LIN {X 0,Y 291.922,Z 233.29,A -85,B 0,C 180,E1 -16667.964,E2 -16667.964} C_VEL
LIN {X 0,Y 291.251,Z 221.348,A -85,B 0,C 180,E1 -16668.598,E2 -16668.598} C_VEL
LIN {X 0,Y 291.234,Z 220.005,A -85,B 0,C 180,E1 -16668.691,E2 -16668.691} C_VEL
LIN {X 0,Y 292.711,Z 208.587,A -85,B 0,C 180,E1 -16673.336,E2 -16673.336} C_VEL
LIN {X 0,Y 294.65,Z 197.089,A -85,B 0,C 180,E1 -16678.051,E2 -16678.051} C_VEL
LIN {X 0,Y 294.841,Z 194.228,A -85,B 0,C 180,E1 -16679.249,E2 -16679.249} C_VEL
LIN {X 0,Y 293.186,Z 185.832,A -85,B 0,C 180,E1 -16682.966,E2 -16682.966} C_VEL
LIN {X 0,Y 291.437,Z 176.187,A -85,B 0,C 180,E1 -16687.432,E2 -16687.432} C_VEL
LIN {X 0,Y 291.323,Z 176.194,A -85,B 0,C 180,E1 -16691.595,E2 -16691.595} C_VEL
LIN {X 0,Y 291.344,Z 176.191,A -85,B 0,C 180,E1 -16695.608,E2 -16695.608} C_VEL
LIN {X 0,Y 291.392,Z 176.185,A -85,B 0,C 180,E1 -16699.367,E2 -16699.367} C_VEL
LIN {X 0,Y 291.423,Z 176.182,A -85,B 0,C 180,E1 -16702.922,E2 -16702.922} C_VEL
LIN {X 0,Y 291.334,Z 176.196,A -85,B 0,C 180,E1 -16706.3,E2 -16706.3} C_VEL
LIN {X 0,Y 291.375,Z 176.19,A -85,B 0,C 180,E1 -16710.259,E2 -16710.259} C_VEL
LIN {X 0,Y 291.404,Z 176.185,A -85,B 0,C 180,E1 -16714.271,E2 -16714.271} C_VEL
LIN {X 0,Y 291.362,Z 176.19,A -85,B 0,C 180,E1 -16717.298,E2 -16717.298} C_VEL
LIN {X 0,Y 291.445,Z 176.179,A -85,B 0,C 180,E1 -16720.269,E2 -16720.269} C_VEL
LIN {X 0,Y 291.542,Z 176.166,A -85,B 0,C 180,E1 -16724.623,E2 -16724.623} C_VEL
LIN {X 0,Y 291.524,Z 176.17,A -85,B 0,C 180,E1 -16728.88,E2 -16728.88} C_VEL
LIN {X 0,Y 291.693,Z 176.149,A -85,B 0,C 180,E1 -16731.688,E2 -16731.688} C_VEL
LIN {X 0,Y 291.618,Z 176.157,A -85,B 0,C 180,E1 -16734.468,E2 -16734.468} C_VEL
LIN {X 0,Y 291.88,Z 176.126,A -85,B 0,C 180,E1 -16738.62,E2 -16738.62} C_VEL
LIN {X 0,Y 291.874,Z 176.127,A -85,B 0,C 180,E1 -16741.38,E2 -16741.38} C_VEL
LIN {X 0,Y 291.732,Z 176.146,A -85,B 0,C 180,E1 -16746.918,E2 -16746.918} C_VEL
LIN {X 0,Y 291.616,Z 176.157,A -85,B 0,C 180,E1 -16749.712,E2 -16749.712} C_VEL
LIN {X 0,Y 291.509,Z 176.172,A -85,B 0,C 180,E1 -16753.951,E2 -16753.951} C_VEL
LIN {X 0,Y 291.474,Z 176.176,A -85,B 0,C 180,E1 -16756.819,E2 -16756.819} C_VEL
LIN {X 0,Y 291.438,Z 176.181,A -85,B 0,C 180,E1 -16759.876,E2 -16759.876} C_VEL
LIN {X 0,Y 291.355,Z 176.194,A -85,B 0,C 180,E1 -16764.209,E2 -16764.209} C_VEL
LIN {X 0,Y 291.346,Z 176.191,A -85,B 0,C 180,E1 -16767.279,E2 -16767.279} C_VEL
LIN {X 0,Y 291.308,Z 176.197,A -85,B 0,C 180,E1 -16770.44,E2 -16770.44} C_VEL
LIN {X 0,Y 291.332,Z 176.196,A -85,B 0,C 180,E1 -16773.7,E2 -16773.7} C_VEL
LIN {X 0,Y 291.383,Z 176.188,A -85,B 0,C 180,E1 -16777.26,E2 -16777.26} C_VEL
LIN {X 0,Y 291.34,Z 176.191,A -85,B 0,C 180,E1 -16780.641,E2 -16780.641} C_VEL
LIN {X 0,Y 291.313,Z 176.195,A -85,B 0,C 180,E1 -16784.398,E2 -16784.398} C_VEL
LIN {X 0,Y 291.318,Z 176.194,A -85,B 0,C 180,E1 -16788.406,E2 -16788.406} C_VEL
LIN {X 0,Y 291.345,Z 176.194,A -85,B 0,C 180,E1 -16791.16,E2 -16791.16} C_VEL
LIN {X 0,Y 291.354,Z 176.191,A -85,B 0,C 180,E1 -16794.628,E2 -16794.628} C_VEL
LIN {X 0,Y 291.366,Z 176.188,A -85,B 0,C 180,E1 -16797.953,E2 -16797.953} C_VEL
LIN {X 0,Y 291.378,Z 176.19,A -85,B 0,C 180,E1 -16801.161,E2 -16801.161} C_VEL
LIN {X 0,Y 291.412,Z 176.184,A -85,B 0,C 180,E1 -16804.274,E2 -16804.274} C_VEL
LIN {X 0,Y 291.378,Z 176.187,A -85,B 0,C 180,E1 -16807.302,E2 -16807.302} C_VEL
LIN {X 0,Y 291.455,Z 176.179,A -85,B 0,C 180,E1 -16810.273,E2 -16810.273} C_VEL
LIN {X 0,Y 291.553,Z 176.169,A -85,B 0,C 180,E1 -16814.626,E2 -16814.626} C_VEL
LIN {X 0,Y 291.536,Z 176.168,A -85,B 0,C 180,E1 -16818.883,E2 -16818.883} C_VEL
LIN {X 0,Y 291.709,Z 176.147,A -85,B 0,C 180,E1 -16821.691,E2 -16821.691} C_VEL
LIN {X 0,Y 291.632,Z 176.157,A -85,B 0,C 180,E1 -16824.471,E2 -16824.471} C_VEL
LIN {X 0,Y 291.878,Z 176.126,A -85,B 0,C 180,E1 -16828.622,E2 -16828.622} C_VEL
LIN {X 0,Y 291.877,Z 176.126,A -85,B 0,C 180,E1 -16831.382,E2 -16831.382} C_VEL
LIN {X 0,Y 291.749,Z 176.141,A -85,B 0,C 180,E1 -16836.92,E2 -16836.92} C_VEL
LIN {X 0,Y 291.632,Z 176.16,A -85,B 0,C 180,E1 -16839.714,E2 -16839.714} C_VEL
LIN {X 0,Y 291.526,Z 176.17,A -85,B 0,C 180,E1 -16843.952,E2 -16843.952} C_VEL
LIN {X 0,Y 291.491,Z 176.174,A -85,B 0,C 180,E1 -16846.82,E2 -16846.82} C_VEL
LIN {X 0,Y 291.455,Z 176.178,A -85,B 0,C 180,E1 -16849.877,E2 -16849.877} C_VEL
LIN {X 0,Y 291.33,Z 176.193,A -85,B 0,C 180,E1 -16854.214,E2 -16854.214} C_VEL
LIN {X 0,Y 291.354,Z 176.193,A -85,B 0,C 180,E1 -16857.281,E2 -16857.281} C_VEL
LIN {X 0,Y 291.323,Z 176.194,A -85,B 0,C 180,E1 -16860.441,E2 -16860.441} C_VEL
LIN {X 0,Y 291.349,Z 176.191,A -85,B 0,C 180,E1 -16863.7,E2 -16863.7} C_VEL
LIN {X 0,Y 291.373,Z 176.188,A -85,B 0,C 180,E1 -16867.253,E2 -16867.253} C_VEL
LIN {X 0,Y 291.305,Z 176.201,A -85,B 0,C 180,E1 -16870.649,E2 -16870.649} C_VEL
LIN {X 0,Y 291.288,Z 176.202,A -85,B 0,C 180,E1 -16874.405,E2 -16874.405} C_VEL
LIN {X 0,Y 291.353,Z 176.195,A -85,B 0,C 180,E1 -16878.401,E2 -16878.401} C_VEL
LIN {X 0,Y 291.346,Z 176.191,A -85,B 0,C 180,E1 -16881.157,E2 -16881.157} C_VEL
LIN {X 0,Y 291.506,Z 176.256,A -85,B 0,C 180,E1 -16885.059,E2 -16885.059} C_VEL
LIN {X 0,Y 292.388,Z 181.277,A -85,B 0,C 180,E1 -16888.075,E2 -16888.075} C_VEL
LIN {X 0,Y 292.465,Z 184.403,A -85,B 0,C 180,E1 -16889.896,E2 -16889.896} C_VEL
LIN {X 0,Y 291.785,Z 191.023,A -85,B 0,C 180,E1 -16893.632,E2 -16893.632} C_VEL
LIN {X 0,Y 291.087,Z 198.926,A -85,B 0,C 180,E1 -16898.023,E2 -16898.023} C_VEL
LIN {X 0,Y 290.624,Z 205.588,A -85,B 0,C 180,E1 -16901.677,E2 -16901.677} C_VEL
LIN {X 0,Y 290.148,Z 213.535,A -85,B 0,C 180,E1 -16905.982,E2 -16905.982} C_VEL
LIN {X 0,Y 290.064,Z 216.758,A -85,B 0,C 180,E1 -16907.627,E2 -16907.627} C_VEL
LIN {X 0,Y 290.735,Z 227.966,A -85,B 0,C 180,E1 -16908.496,E2 -16908.496} C_VEL
LIN {X 0,Y 291.517,Z 238.59,A -85,B 0,C 180,E1 -16909.583,E2 -16909.583} C_VEL
LIN {X 0,Y 291.006,Z 247.91,A -85,B 0,C 180,E1 -16910.793,E2 -16910.793} C_VEL
LIN {X 0,Y 290.536,Z 257.449,A -85,B 0,C 180,E1 -16912.355,E2 -16912.355} C_VEL
LIN {X 0,Y 290.137,Z 266.131,A -85,B 0,C 180,E1 -16914.18,E2 -16914.18} C_VEL
LIN {X 0,Y 289.948,Z 272.322,A -85,B 0,C 180,E1 -16915.83,E2 -16915.83} C_VEL
LIN {X 0,Y 289.63,Z 278.288,A -85,B 0,C 180,E1 -16917.914,E2 -16917.914} C_VEL
LIN {X 0,Y 289.621,Z 282.573,A -85,B 0,C 180,E1 -16920,E2 -16920} C_VEL
LIN {X 0,Y 289.778,Z 284.578,A -85,B 0,C 180,E1 -16921.39,E2 -16921.39} C_VEL
LIN {X 0,Y 290.075,Z 285.942,A -85,B 0,C 180,E1 -16922.778,E2 -16922.778} C_VEL
LIN {X 0,Y 290.874,Z 286.751,A -85,B 0,C 180,E1 -16924.841,E2 -16924.841} C_VEL
LIN {X 0,Y 290.556,Z 286.874,A -85,B 0,C 180,E1 -16925.623,E2 -16925.623} C_VEL
LIN {X 0,Y 288.243,Z 286.846,A -85,B 0,C 180,E1 -16926.881,E2 -16926.881} C_VEL
LIN {X 0,Y 285.999,Z 286.418,A -85,B 0,C 180,E1 -16928.153,E2 -16928.153} C_VEL
LIN {X 0,Y 285.799,Z 285.781,A -85,B 0,C 180,E1 -16928.941,E2 -16928.941} C_VEL
LIN {X 0,Y 287.146,Z 283.854,A -85,B 0,C 180,E1 -16930.578,E2 -16930.578} C_VEL
LIN {X 0,Y 289.141,Z 280.078,A -85,B 0,C 180,E1 -16932.636,E2 -16932.636} C_VEL
LIN {X 0,Y 291.713,Z 274.767,A -85,B 0,C 180,E1 -16934.653,E2 -16934.653} C_VEL
LIN {X 0,Y 294.634,Z 267.761,A -85,B 0,C 180,E1 -16936.633,E2 -16936.633} C_VEL
LIN {X 0,Y 296.937,Z 260.933,A -85,B 0,C 180,E1 -16938.173,E2 -16938.173} C_VEL
LIN {X 0,Y 297.396,Z 254.438,A -85,B 0,C 180,E1 -16939.679,E2 -16939.679} C_VEL
LIN {X 0,Y 297.034,Z 246.793,A -85,B 0,C 180,E1 -16941.399,E2 -16941.399} C_VEL
LIN {X 0,Y 295.632,Z 237.751,A -85,B 0,C 180,E1 -16943.44,E2 -16943.44} C_VEL
LIN {X 0,Y 293.399,Z 228.753,A -85,B 0,C 180,E1 -16945.542,E2 -16945.542} C_VEL
LIN {X 0,Y 290.202,Z 219.279,A -85,B 0,C 180,E1 -16947.984,E2 -16947.984} C_VEL
LIN {X 0,Y 290.597,Z 218.071,A -85,B 0,C 180,E1 -16948.927,E2 -16948.927} C_VEL
LIN {X 0,Y 292.066,Z 214.685,A -85,B 0,C 180,E1 -16952.623,E2 -16952.623} C_VEL
LIN {X 0,Y 292.453,Z 212.978,A -85,B 0,C 180,E1 -16955.223,E2 -16955.223} C_VEL
LIN {X 0,Y 292.573,Z 211.549,A -85,B 0,C 180,E1 -16958.65,E2 -16958.65} C_VEL
LIN {X 0,Y 292.684,Z 210.994,A -85,B 0,C 180,E1 -16962.248,E2 -16962.248} C_VEL
LIN {X 0,Y 293.006,Z 211.385,A -85,B 0,C 180,E1 -16966.02,E2 -16966.02} C_VEL
LIN {X 0,Y 293.322,Z 212.845,A -85,B 0,C 180,E1 -16969.688,E2 -16969.688} C_VEL
LIN {X 0,Y 293.711,Z 215.311,A -85,B 0,C 180,E1 -16973.256,E2 -16973.256} C_VEL
LIN {X 0,Y 294.042,Z 216.854,A -85,B 0,C 180,E1 -16974.994,E2 -16974.994} C_VEL
LIN {X 0,Y 294.515,Z 220.412,A -85,B 0,C 180,E1 -16978.166,E2 -16978.166} C_VEL
LIN {X 0,Y 296.581,Z 225.556,A -85,B 0,C 180,E1 -16979.265,E2 -16979.265} C_VEL
LIN {X 0,Y 298.966,Z 236.054,A -85,B 0,C 180,E1 -16981.041,E2 -16981.041} C_VEL
LIN {X 0,Y 300.396,Z 246.753,A -85,B 0,C 180,E1 -16982.753,E2 -16982.753} C_VEL
LIN {X 0,Y 300.603,Z 256.384,A -85,B 0,C 180,E1 -16984.261,E2 -16984.261} C_VEL
LIN {X 0,Y 299.872,Z 262.807,A -85,B 0,C 180,E1 -16985.231,E2 -16985.231} C_VEL
LIN {X 0,Y 297.025,Z 272.375,A -85,B 0,C 180,E1 -16986.649,E2 -16986.649} C_VEL
LIN {X 0,Y 294.133,Z 281.208,A -85,B 0,C 180,E1 -16988.26,E2 -16988.26} C_VEL
LIN {X 0,Y 291.061,Z 289.915,A -85,B 0,C 180,E1 -16990.24,E2 -16990.24} C_VEL
LIN {X 0,Y 288.565,Z 296.948,A -85,B 0,C 180,E1 -16992.274,E2 -16992.274} C_VEL
LIN {X 0,Y 286.676,Z 302.672,A -85,B 0,C 180,E1 -16994.353,E2 -16994.353} C_VEL
LIN {X 0,Y 284.897,Z 307.26,A -85,B 0,C 180,E1 -16996.445,E2 -16996.445} C_VEL
LIN {X 0,Y 283.731,Z 310.784,A -85,B 0,C 180,E1 -16998.569,E2 -16998.569} C_VEL
LIN {X 0,Y 282.79,Z 313.971,A -85,B 0,C 180,E1 -17001.422,E2 -17001.422} C_VEL
LIN {X 0,Y 282.552,Z 314.982,A -85,B 0,C 180,E1 -17002.854,E2 -17002.854} C_VEL
LIN {X 0,Y 282.488,Z 315.573,A -85,B 0,C 180,E1 -17004.362,E2 -17004.362} C_VEL
LIN {X 0,Y 282.48,Z 315.734,A -85,B 0,C 180,E1 -17005.717,E2 -17005.717} C_VEL
LIN {X 0,Y 282.487,Z 315.516,A -85,B 0,C 180,E1 -17007.146,E2 -17007.146} C_VEL
LIN {X 0,Y 282.811,Z 314.871,A -85,B 0,C 180,E1 -17008.574,E2 -17008.574} C_VEL
LIN {X 0,Y 282.89,Z 313.769,A -85,B 0,C 180,E1 -17009.998,E2 -17009.998} C_VEL
LIN {X 0,Y 282.885,Z 311.242,A -85,B 0,C 180,E1 -17012.133,E2 -17012.133} C_VEL
LIN {X 0,Y 282.838,Z 307.581,A -85,B 0,C 180,E1 -17014.273,E2 -17014.273} C_VEL
LIN {X 0,Y 282.952,Z 302.371,A -85,B 0,C 180,E1 -17016.52,E2 -17016.52} C_VEL
LIN {X 0,Y 283.084,Z 296.24,A -85,B 0,C 180,E1 -17018.564,E2 -17018.564} C_VEL
LIN {X 0,Y 283.332,Z 289.589,A -85,B 0,C 180,E1 -17020.358,E2 -17020.358} C_VEL
LIN {X 0,Y 283.815,Z 281.5,A -85,B 0,C 180,E1 -17022.148,E2 -17022.148} C_VEL
LIN {X 0,Y 284.51,Z 271.428,A -85,B 0,C 180,E1 -17023.934,E2 -17023.934} C_VEL
LIN {X 0,Y 285.137,Z 261.442,A -85,B 0,C 180,E1 -17025.362,E2 -17025.362} C_VEL
LIN {X 0,Y 285.939,Z 250.048,A -85,B 0,C 180,E1 -17026.642,E2 -17026.642} C_VEL
LIN {X 0,Y 285.956,Z 246.019,A -85,B 0,C 180,E1 -17027.023,E2 -17027.023} C_VEL
LIN {X 0,Y 284.874,Z 234.213,A -85,B 0,C 180,E1 -17027.959,E2 -17027.959} C_VEL
LIN {X 0,Y 284.188,Z 222.921,A -85,B 0,C 180,E1 -17028.61,E2 -17028.61} C_VEL
LIN {X 0,Y 284.168,Z 220.049,A -85,B 0,C 180,E1 -17028.752,E2 -17028.752} C_VEL
LIN {X 0,Y 285.522,Z 209.459,A -85,B 0,C 180,E1 -17033.19,E2 -17033.19} C_VEL
LIN {X 0,Y 287.384,Z 198.799,A -85,B 0,C 180,E1 -17037.684,E2 -17037.684} C_VEL
LIN {X 0,Y 287.805,Z 195.191,A -85,B 0,C 180,E1 -17039.232,E2 -17039.232} C_VEL
LIN {X 0,Y 286.013,Z 186.137,A -85,B 0,C 180,E1 -17043.336,E2 -17043.336} C_VEL
LIN {X 0,Y 284.369,Z 177.068,A -85,B 0,C 180,E1 -17047.687,E2 -17047.687} C_VEL
LIN {X 0,Y 284.275,Z 177.073,A -85,B 0,C 180,E1 -17052.125,E2 -17052.125} C_VEL
LIN {X 0,Y 284.31,Z 177.07,A -85,B 0,C 180,E1 -17056.199,E2 -17056.199} C_VEL
LIN {X 0,Y 284.342,Z 177.066,A -85,B 0,C 180,E1 -17060.011,E2 -17060.011} C_VEL
LIN {X 0,Y 284.345,Z 177.064,A -85,B 0,C 180,E1 -17063.616,E2 -17063.616} C_VEL
LIN {X 0,Y 284.297,Z 177.069,A -85,B 0,C 180,E1 -17067.188,E2 -17067.188} C_VEL
LIN {X 0,Y 284.347,Z 177.065,A -85,B 0,C 180,E1 -17070.375,E2 -17070.375} C_VEL
LIN {X 0,Y 284.366,Z 177.062,A -85,B 0,C 180,E1 -17073.585,E2 -17073.585} C_VEL
LIN {X 0,Y 284.321,Z 177.066,A -85,B 0,C 180,E1 -17076.703,E2 -17076.703} C_VEL
LIN {X 0,Y 284.39,Z 177.059,A -85,B 0,C 180,E1 -17081.261,E2 -17081.261} C_VEL
LIN {X 0,Y 284.479,Z 177.046,A -85,B 0,C 180,E1 -17084.458,E2 -17084.458} C_VEL
LIN {X 0,Y 284.476,Z 177.047,A -85,B 0,C 180,E1 -17088.601,E2 -17088.601} C_VEL
LIN {X 0,Y 284.643,Z 177.028,A -85,B 0,C 180,E1 -17091.481,E2 -17091.481} C_VEL
LIN {X 0,Y 284.588,Z 177.033,A -85,B 0,C 180,E1 -17094.331,E2 -17094.331} C_VEL
LIN {X 0,Y 284.846,Z 177.002,A -85,B 0,C 180,E1 -17098.586,E2 -17098.586} C_VEL
LIN {X 0,Y 284.84,Z 177.003,A -85,B 0,C 180,E1 -17101.414,E2 -17101.414} C_VEL
LIN {X 0,Y 284.684,Z 177.022,A -85,B 0,C 180,E1 -17107.09,E2 -17107.09} C_VEL
LIN {X 0,Y 284.553,Z 177.037,A -85,B 0,C 180,E1 -17109.956,E2 -17109.956} C_VEL
LIN {X 0,Y 284.469,Z 177.051,A -85,B 0,C 180,E1 -17114.303,E2 -17114.303} C_VEL
LIN {X 0,Y 284.413,Z 177.054,A -85,B 0,C 180,E1 -17117.249,E2 -17117.249} C_VEL
LIN {X 0,Y 284.366,Z 177.064,A -85,B 0,C 180,E1 -17120.243,E2 -17120.243} C_VEL
LIN {X 0,Y 284.314,Z 177.069,A -85,B 0,C 180,E1 -17123.857,E2 -17123.857} C_VEL
LIN {X 0,Y 284.276,Z 177.076,A -85,B 0,C 180,E1 -17128.017,E2 -17128.017} C_VEL
LIN {X 0,Y 284.273,Z 177.073,A -85,B 0,C 180,E1 -17131.277,E2 -17131.277} C_VEL
LIN {X 0,Y 284.351,Z 177.063,A -85,B 0,C 180,E1 -17135.356,E2 -17135.356} C_VEL
LIN {X 0,Y 284.313,Z 177.069,A -85,B 0,C 180,E1 -17138.169,E2 -17138.169} C_VEL
LIN {X 0,Y 284.286,Z 177.07,A -85,B 0,C 180,E1 -17142.132,E2 -17142.132} C_VEL
LIN {X 0,Y 284.26,Z 177.074,A -85,B 0,C 180,E1 -17146.194,E2 -17146.194} C_VEL
LIN {X 0,Y 284.298,Z 177.069,A -85,B 0,C 180,E1 -17150.026,E2 -17150.026} C_VEL
LIN {X 0,Y 284.325,Z 177.067,A -85,B 0,C 180,E1 -17153.616,E2 -17153.616} C_VEL
LIN {X 0,Y 284.301,Z 177.072,A -85,B 0,C 180,E1 -17157.192,E2 -17157.192} C_VEL
LIN {X 0,Y 284.353,Z 177.061,A -85,B 0,C 180,E1 -17160.378,E2 -17160.378} C_VEL
LIN {X 0,Y 284.373,Z 177.06,A -85,B 0,C 180,E1 -17163.589,E2 -17163.589} C_VEL
LIN {X 0,Y 284.363,Z 177.065,A -85,B 0,C 180,E1 -17166.709,E2 -17166.709} C_VEL
LIN {X 0,Y 284.401,Z 177.057,A -85,B 0,C 180,E1 -17171.264,E2 -17171.264} C_VEL
LIN {X 0,Y 284.49,Z 177.05,A -85,B 0,C 180,E1 -17174.461,E2 -17174.461} C_VEL
LIN {X 0,Y 284.487,Z 177.048,A -85,B 0,C 180,E1 -17178.604,E2 -17178.604} C_VEL
LIN {X 0,Y 284.659,Z 177.024,A -85,B 0,C 180,E1 -17181.483,E2 -17181.483} C_VEL
LIN {X 0,Y 284.602,Z 177.034,A -85,B 0,C 180,E1 -17184.334,E2 -17184.334} C_VEL
LIN {X 0,Y 284.846,Z 177.002,A -85,B 0,C 180,E1 -17188.588,E2 -17188.588} C_VEL
LIN {X 0,Y 284.845,Z 177.002,A -85,B 0,C 180,E1 -17191.416,E2 -17191.416} C_VEL
LIN {X 0,Y 284.701,Z 177.019,A -85,B 0,C 180,E1 -17197.092,E2 -17197.092} C_VEL
LIN {X 0,Y 284.57,Z 177.037,A -85,B 0,C 180,E1 -17199.957,E2 -17199.957} C_VEL
LIN {X 0,Y 284.485,Z 177.045,A -85,B 0,C 180,E1 -17204.305,E2 -17204.305} C_VEL
LIN {X 0,Y 284.429,Z 177.056,A -85,B 0,C 180,E1 -17207.25,E2 -17207.25} C_VEL
LIN {X 0,Y 284.38,Z 177.058,A -85,B 0,C 180,E1 -17210.244,E2 -17210.244} C_VEL
LIN {X 0,Y 284.287,Z 177.073,A -85,B 0,C 180,E1 -17214.853,E2 -17214.853} C_VEL
LIN {X 0,Y 284.285,Z 177.07,A -85,B 0,C 180,E1 -17218.018,E2 -17218.018} C_VEL
LIN {X 0,Y 284.29,Z 177.072,A -85,B 0,C 180,E1 -17221.277,E2 -17221.277} C_VEL
LIN {X 0,Y 284.342,Z 177.065,A -85,B 0,C 180,E1 -17225.348,E2 -17225.348} C_VEL
LIN {X 0,Y 284.306,Z 177.068,A -85,B 0,C 180,E1 -17228.172,E2 -17228.172} C_VEL
LIN {X 0,Y 284.242,Z 177.077,A -85,B 0,C 180,E1 -17232.118,E2 -17232.118} C_VEL
LIN {X 0,Y 284.262,Z 177.076,A -85,B 0,C 180,E1 -17236.19,E2 -17236.19} C_VEL
LIN {X 0,Y 284.313,Z 177.069,A -85,B 0,C 180,E1 -17240.025,E2 -17240.025} C_VEL
LIN {X 0,Y 284.437,Z 177.055,A -85,B 0,C 180,E1 -17244.628,E2 -17244.628} C_VEL
LIN {X 0,Y 284.477,Z 177.176,A -85,B 0,C 180,E1 -17245.005,E2 -17245.005} C_VEL
LIN {X 0,Y 285.355,Z 182.094,A -85,B 0,C 180,E1 -17248.027,E2 -17248.027} C_VEL
LIN {X 0,Y 285.462,Z 184.594,A -85,B 0,C 180,E1 -17249.51,E2 -17249.51} C_VEL
LIN {X 0,Y 284.918,Z 190.002,A -85,B 0,C 180,E1 -17252.627,E2 -17252.627} C_VEL
LIN {X 0,Y 284.191,Z 197.115,A -85,B 0,C 180,E1 -17256.692,E2 -17256.692} C_VEL
LIN {X 0,Y 283.715,Z 203.489,A -85,B 0,C 180,E1 -17260.277,E2 -17260.277} C_VEL
LIN {X 0,Y 283.189,Z 210.47,A -85,B 0,C 180,E1 -17264.158,E2 -17264.158} C_VEL
LIN {X 0,Y 283,Z 216.617,A -85,B 0,C 180,E1 -17267.541,E2 -17267.541} C_VEL
LIN {X 0,Y 283.653,Z 228.157,A -85,B 0,C 180,E1 -17268.477,E2 -17268.477} C_VEL
LIN {X 0,Y 284.437,Z 237.98,A -85,B 0,C 180,E1 -17269.501,E2 -17269.501} C_VEL
LIN {X 0,Y 283.903,Z 248.683,A -85,B 0,C 180,E1 -17270.92,E2 -17270.92} C_VEL
LIN {X 0,Y 283.387,Z 258.077,A -85,B 0,C 180,E1 -17272.519,E2 -17272.519} C_VEL
LIN {X 0,Y 283.042,Z 266.311,A -85,B 0,C 180,E1 -17274.3,E2 -17274.3} C_VEL
LIN {X 0,Y 282.815,Z 272.827,A -85,B 0,C 180,E1 -17276.082,E2 -17276.082} C_VEL
LIN {X 0,Y 282.552,Z 277.884,A -85,B 0,C 180,E1 -17277.862,E2 -17277.862} C_VEL
LIN {X 0,Y 282.533,Z 282.42,A -85,B 0,C 180,E1 -17280,E2 -17280} C_VEL
LIN {X 0,Y 282.69,Z 284.584,A -85,B 0,C 180,E1 -17281.425,E2 -17281.425} C_VEL
LIN {X 0,Y 282.992,Z 286.121,A -85,B 0,C 180,E1 -17282.847,E2 -17282.847} C_VEL
LIN {X 0,Y 283.491,Z 287.052,A -85,B 0,C 180,E1 -17284.265,E2 -17284.265} C_VEL
LIN {X 0,Y 284.199,Z 287.358,A -85,B 0,C 180,E1 -17285.677,E2 -17285.677} C_VEL
LIN {X 0,Y 284.689,Z 287.086,A -85,B 0,C 180,E1 -17287.09,E2 -17287.09} C_VEL
LIN {X 0,Y 285.799,Z 285.781,A -85,B 0,C 180,E1 -17288.941,E2 -17288.941} C_VEL
LIN {X 0,Y 285.691,Z 285.122,A -85,B 0,C 180,E1 -17289.734,E2 -17289.734} C_VEL
LIN {X 0,Y 282.327,Z 282.599,A -85,B 0,C 180,E1 -17292.33,E2 -17292.33} C_VEL
LIN {X 0,Y 282.538,Z 281.272,A -85,B 0,C 180,E1 -17293.086,E2 -17293.086} C_VEL
LIN {X 0,Y 285.045,Z 276.665,A -85,B 0,C 180,E1 -17295.004,E2 -17295.004} C_VEL
LIN {X 0,Y 288.099,Z 270.13,A -85,B 0,C 180,E1 -17297.022,E2 -17297.022} C_VEL
LIN {X 0,Y 290.746,Z 263.4,A -85,B 0,C 180,E1 -17298.654,E2 -17298.654} C_VEL
LIN {X 0,Y 291.479,Z 256.132,A -85,B 0,C 180,E1 -17300.463,E2 -17300.463} C_VEL
LIN {X 0,Y 291.291,Z 248.612,A -85,B 0,C 180,E1 -17302.287,E2 -17302.287} C_VEL
LIN {X 0,Y 290.188,Z 240.323,A -85,B 0,C 180,E1 -17304.313,E2 -17304.313} C_VEL
LIN {X 0,Y 288.364,Z 232.193,A -85,B 0,C 180,E1 -17306.41,E2 -17306.41} C_VEL
LIN {X 0,Y 286.087,Z 224.218,A -85,B 0,C 180,E1 -17308.622,E2 -17308.622} C_VEL
LIN {X 0,Y 284.723,Z 220.89,A -85,B 0,C 180,E1 -17309.733,E2 -17309.733} C_VEL
LIN {X 0,Y 284.378,Z 219.142,A -85,B 0,C 180,E1 -17310.236,E2 -17310.236} C_VEL
LIN {X 0,Y 285.458,Z 216.716,A -85,B 0,C 180,E1 -17313.164,E2 -17313.164} C_VEL
LIN {X 0,Y 285.828,Z 215.025,A -85,B 0,C 180,E1 -17316.166,E2 -17316.166} C_VEL
LIN {X 0,Y 285.928,Z 214.262,A -85,B 0,C 180,E1 -17318.133,E2 -17318.133} C_VEL
LIN {X 0,Y 286.043,Z 213.65,A -85,B 0,C 180,E1 -17321.559,E2 -17321.559} C_VEL
LIN {X 0,Y 286.337,Z 213.883,A -85,B 0,C 180,E1 -17325.381,E2 -17325.381} C_VEL
LIN {X 0,Y 286.589,Z 214.93,A -85,B 0,C 180,E1 -17328.536,E2 -17328.536} C_VEL
LIN {X 0,Y 286.995,Z 217.115,A -85,B 0,C 180,E1 -17332.249,E2 -17332.249} C_VEL
LIN {X 0,Y 287.243,Z 218.52,A -85,B 0,C 180,E1 -17334.038,E2 -17334.038} C_VEL
LIN {X 0,Y 287.531,Z 220.433,A -85,B 0,C 180,E1 -17335.912,E2 -17335.912} C_VEL
LIN {X 0,Y 289.002,Z 223.556,A -85,B 0,C 180,E1 -17336.801,E2 -17336.801} C_VEL
LIN {X 0,Y 290.855,Z 226.417,A -85,B 0,C 180,E1 -17337.749,E2 -17337.749} C_VEL
LIN {X 0,Y 292.337,Z 230.74,A -85,B 0,C 180,E1 -17338.724,E2 -17338.724} C_VEL
LIN {X 0,Y 294.003,Z 239.669,A -85,B 0,C 180,E1 -17340.356,E2 -17340.356} C_VEL
LIN {X 0,Y 294.981,Z 250.459,A -85,B 0,C 180,E1 -17342.21,E2 -17342.21} C_VEL
LIN {X 0,Y 294.835,Z 259.143,A -85,B 0,C 180,E1 -17343.672,E2 -17343.672} C_VEL
LIN {X 0,Y 294.024,Z 264.385,A -85,B 0,C 180,E1 -17344.514,E2 -17344.514} C_VEL
LIN {X 0,Y 290.713,Z 274.484,A -85,B 0,C 180,E1 -17346.111,E2 -17346.111} C_VEL
LIN {X 0,Y 287.117,Z 284.315,A -85,B 0,C 180,E1 -17348.079,E2 -17348.079} C_VEL
LIN {X 0,Y 283.879,Z 292.575,A -85,B 0,C 180,E1 -17350.181,E2 -17350.181} C_VEL
LIN {X 0,Y 281.17,Z 299.723,A -85,B 0,C 180,E1 -17352.543,E2 -17352.543} C_VEL
LIN {X 0,Y 279.192,Z 304.781,A -85,B 0,C 180,E1 -17354.672,E2 -17354.672} C_VEL
LIN {X 0,Y 277.478,Z 308.764,A -85,B 0,C 180,E1 -17356.821,E2 -17356.821} C_VEL
LIN {X 0,Y 276.162,Z 312.519,A -85,B 0,C 180,E1 -17359.736,E2 -17359.736} C_VEL
LIN {X 0,Y 275.732,Z 313.804,A -85,B 0,C 180,E1 -17361.201,E2 -17361.201} C_VEL
LIN {X 0,Y 275.392,Z 315.135,A -85,B 0,C 180,E1 -17364.139,E2 -17364.139} C_VEL
LIN {X 0,Y 275.401,Z 315.223,A -85,B 0,C 180,E1 -17365.607,E2 -17365.607} C_VEL
LIN {X 0,Y 275.414,Z 314.858,A -85,B 0,C 180,E1 -17367.072,E2 -17367.072} C_VEL
LIN {X 0,Y 275.749,Z 314.114,A -85,B 0,C 180,E1 -17368.537,E2 -17368.537} C_VEL
LIN {X 0,Y 275.84,Z 312.928,A -85,B 0,C 180,E1 -17369.998,E2 -17369.998} C_VEL
LIN {X 0,Y 275.855,Z 310.221,A -85,B 0,C 180,E1 -17372.188,E2 -17372.188} C_VEL
LIN {X 0,Y 275.839,Z 306.336,A -85,B 0,C 180,E1 -17374.381,E2 -17374.381} C_VEL
LIN {X 0,Y 275.932,Z 301.068,A -85,B 0,C 180,E1 -17376.619,E2 -17376.619} C_VEL
LIN {X 0,Y 276.069,Z 294.528,A -85,B 0,C 180,E1 -17378.784,E2 -17378.784} C_VEL
LIN {X 0,Y 276.442,Z 286.025,A -85,B 0,C 180,E1 -17380.99,E2 -17380.99} C_VEL
LIN {X 0,Y 276.948,Z 277.211,A -85,B 0,C 180,E1 -17382.827,E2 -17382.827} C_VEL
LIN {X 0,Y 277.559,Z 268.569,A -85,B 0,C 180,E1 -17384.29,E2 -17384.29} C_VEL
LIN {X 0,Y 278.298,Z 257.965,A -85,B 0,C 180,E1 -17385.749,E2 -17385.749} C_VEL
LIN {X 0,Y 278.952,Z 248.24,A -85,B 0,C 180,E1 -17386.821,E2 -17386.821} C_VEL
LIN {X 0,Y 277.94,Z 236.194,A -85,B 0,C 180,E1 -17387.851,E2 -17387.851} C_VEL
LIN {X 0,Y 277.142,Z 223.946,A -85,B 0,C 180,E1 -17388.622,E2 -17388.622} C_VEL
LIN {X 0,Y 277.097,Z 219.923,A -85,B 0,C 180,E1 -17388.865,E2 -17388.865} C_VEL
LIN {X 0,Y 278.656,Z 208.529,A -85,B 0,C 180,E1 -17393.797,E2 -17393.797} C_VEL
LIN {X 0,Y 280.582,Z 197.88,A -85,B 0,C 180,E1 -17398.416,E2 -17398.416} C_VEL
LIN {X 0,Y 280.71,Z 195.779,A -85,B 0,C 180,E1 -17399.346,E2 -17399.346} C_VEL
LIN {X 0,Y 279.255,Z 188.492,A -85,B 0,C 180,E1 -17402.755,E2 -17402.755} C_VEL
LIN {X 0,Y 277.498,Z 178.813,A -85,B 0,C 180,E1 -17407.429,E2 -17407.429} C_VEL
LIN {X 0,Y 277.304,Z 177.949,A -85,B 0,C 180,E1 -17407.964,E2 -17407.964} C_VEL
LIN {X 0,Y 277.225,Z 177.954,A -85,B 0,C 180,E1 -17412.677,E2 -17412.677} C_VEL
LIN {X 0,Y 277.254,Z 177.947,A -85,B 0,C 180,E1 -17416.81,E2 -17416.81} C_VEL
LIN {X 0,Y 277.258,Z 177.948,A -85,B 0,C 180,E1 -17420.676,E2 -17420.676} C_VEL
LIN {X 0,Y 277.295,Z 177.944,A -85,B 0,C 180,E1 -17424.343,E2 -17424.343} C_VEL
LIN {X 0,Y 277.234,Z 177.951,A -85,B 0,C 180,E1 -17427.835,E2 -17427.835} C_VEL
LIN {X 0,Y 277.26,Z 177.946,A -85,B 0,C 180,E1 -17431.209,E2 -17431.209} C_VEL
LIN {X 0,Y 277.298,Z 177.941,A -85,B 0,C 180,E1 -17434.478,E2 -17434.478} C_VEL
LIN {X 0,Y 277.256,Z 177.95,A -85,B 0,C 180,E1 -17437.652,E2 -17437.652} C_VEL
LIN {X 0,Y 277.332,Z 177.937,A -85,B 0,C 180,E1 -17440.765,E2 -17440.765} C_VEL
LIN {X 0,Y 277.422,Z 177.928,A -85,B 0,C 180,E1 -17445.325,E2 -17445.325} C_VEL
LIN {X 0,Y 277.494,Z 177.917,A -85,B 0,C 180,E1 -17449.788,E2 -17449.788} C_VEL
LIN {X 0,Y 277.636,Z 177.899,A -85,B 0,C 180,E1 -17452.729,E2 -17452.729} C_VEL
LIN {X 0,Y 277.812,Z 177.878,A -85,B 0,C 180,E1 -17458.55,E2 -17458.55} C_VEL
LIN {X 0,Y 277.806,Z 177.879,A -85,B 0,C 180,E1 -17461.45,E2 -17461.45} C_VEL
LIN {X 0,Y 277.639,Z 177.899,A -85,B 0,C 180,E1 -17467.271,E2 -17467.271} C_VEL
LIN {X 0,Y 277.494,Z 177.917,A -85,B 0,C 180,E1 -17470.212,E2 -17470.212} C_VEL
LIN {X 0,Y 277.422,Z 177.929,A -85,B 0,C 180,E1 -17474.675,E2 -17474.675} C_VEL
LIN {X 0,Y 277.334,Z 177.936,A -85,B 0,C 180,E1 -17479.235,E2 -17479.235} C_VEL
LIN {X 0,Y 277.275,Z 177.946,A -85,B 0,C 180,E1 -17483.925,E2 -17483.925} C_VEL
LIN {X 0,Y 277.261,Z 177.946,A -85,B 0,C 180,E1 -17487.486,E2 -17487.486} C_VEL
LIN {X 0,Y 277.236,Z 177.95,A -85,B 0,C 180,E1 -17490.474,E2 -17490.474} C_VEL
LIN {X 0,Y 277.242,Z 177.951,A -85,B 0,C 180,E1 -17493.896,E2 -17493.896} C_VEL
LIN {X 0,Y 277.27,Z 177.947,A -85,B 0,C 180,E1 -17497.469,E2 -17497.469} C_VEL
LIN {X 0,Y 277.217,Z 177.953,A -85,B 0,C 180,E1 -17501.235,E2 -17501.235} C_VEL
LIN {X 0,Y 277.211,Z 177.954,A -85,B 0,C 180,E1 -17505.224,E2 -17505.224} C_VEL
LIN {X 0,Y 277.215,Z 177.954,A -85,B 0,C 180,E1 -17509.514,E2 -17509.514} C_VEL
LIN {X 0,Y 277.26,Z 177.945,A -85,B 0,C 180,E1 -17512.533,E2 -17512.533} C_VEL
LIN {X 0,Y 277.24,Z 177.948,A -85,B 0,C 180,E1 -17516.107,E2 -17516.107} C_VEL
LIN {X 0,Y 277.256,Z 177.946,A -85,B 0,C 180,E1 -17519.541,E2 -17519.541} C_VEL
LIN {X 0,Y 277.354,Z 177.938,A -85,B 0,C 180,E1 -17522.867,E2 -17522.867} C_VEL
LIN {X 0,Y 277.325,Z 177.938,A -85,B 0,C 180,E1 -17526.082,E2 -17526.082} C_VEL
LIN {X 0,Y 277.342,Z 177.939,A -85,B 0,C 180,E1 -17530.769,E2 -17530.769} C_VEL
LIN {X 0,Y 277.433,Z 177.924,A -85,B 0,C 180,E1 -17535.328,E2 -17535.328} C_VEL
LIN {X 0,Y 277.506,Z 177.916,A -85,B 0,C 180,E1 -17539.791,E2 -17539.791} C_VEL
LIN {X 0,Y 277.654,Z 177.898,A -85,B 0,C 180,E1 -17542.732,E2 -17542.732} C_VEL
LIN {X 0,Y 277.813,Z 177.878,A -85,B 0,C 180,E1 -17548.553,E2 -17548.553} C_VEL
LIN {X 0,Y 277.812,Z 177.878,A -85,B 0,C 180,E1 -17551.452,E2 -17551.452} C_VEL
LIN {X 0,Y 277.656,Z 177.898,A -85,B 0,C 180,E1 -17557.273,E2 -17557.273} C_VEL
LIN {X 0,Y 277.51,Z 177.915,A -85,B 0,C 180,E1 -17560.213,E2 -17560.213} C_VEL
LIN {X 0,Y 277.438,Z 177.923,A -85,B 0,C 180,E1 -17564.676,E2 -17564.676} C_VEL
LIN {X 0,Y 277.349,Z 177.938,A -85,B 0,C 180,E1 -17569.236,E2 -17569.236} C_VEL
LIN {X 0,Y 277.259,Z 177.946,A -85,B 0,C 180,E1 -17573.929,E2 -17573.929} C_VEL
LIN {X 0,Y 277.271,Z 177.946,A -85,B 0,C 180,E1 -17577.483,E2 -17577.483} C_VEL
LIN {X 0,Y 277.253,Z 177.946,A -85,B 0,C 180,E1 -17580.474,E2 -17580.474} C_VEL
LIN {X 0,Y 277.251,Z 177.947,A -85,B 0,C 180,E1 -17583.897,E2 -17583.897} C_VEL
LIN {X 0,Y 277.265,Z 177.944,A -85,B 0,C 180,E1 -17587.472,E2 -17587.472} C_VEL
LIN {X 0,Y 277.189,Z 177.955,A -85,B 0,C 180,E1 -17591.243,E2 -17591.243} C_VEL
LIN {X 0,Y 277.204,Z 177.953,A -85,B 0,C 180,E1 -17595.228,E2 -17595.228} C_VEL
LIN {X 0,Y 277.226,Z 177.952,A -85,B 0,C 180,E1 -17598.766,E2 -17598.766} C_VEL
LIN {X 0,Y 277.283,Z 177.945,A -85,B 0,C 180,E1 -17602.533,E2 -17602.533} C_VEL
LIN {X 0,Y 277.405,Z 178.04,A -85,B 0,C 180,E1 -17604.916,E2 -17604.916} C_VEL
LIN {X 0,Y 278.298,Z 182.904,A -85,B 0,C 180,E1 -17607.973,E2 -17607.973} C_VEL
LIN {X 0,Y 278.365,Z 185.703,A -85,B 0,C 180,E1 -17609.672,E2 -17609.672} C_VEL
LIN {X 0,Y 277.794,Z 191.194,A -85,B 0,C 180,E1 -17612.91,E2 -17612.91} C_VEL
LIN {X 0,Y 276.98,Z 199.319,A -85,B 0,C 180,E1 -17617.629,E2 -17617.629} C_VEL
LIN {X 0,Y 276.455,Z 206.021,A -85,B 0,C 180,E1 -17621.472,E2 -17621.472} C_VEL
LIN {X 0,Y 275.967,Z 214.125,A -85,B 0,C 180,E1 -17626.058,E2 -17626.058} C_VEL
LIN {X 0,Y 275.919,Z 216.679,A -85,B 0,C 180,E1 -17627.496,E2 -17627.496} C_VEL
LIN {X 0,Y 276.552,Z 228.21,A -85,B 0,C 180,E1 -17628.456,E2 -17628.456} C_VEL
LIN {X 0,Y 277.286,Z 238.792,A -85,B 0,C 180,E1 -17629.596,E2 -17629.596} C_VEL
LIN {X 0,Y 276.76,Z 249.322,A -85,B 0,C 180,E1 -17631.052,E2 -17631.052} C_VEL
LIN {X 0,Y 276.255,Z 258.627,A -85,B 0,C 180,E1 -17632.692,E2 -17632.692} C_VEL
LIN {X 0,Y 275.954,Z 266.803,A -85,B 0,C 180,E1 -17634.52,E2 -17634.52} C_VEL
LIN {X 0,Y 275.687,Z 273.272,A -85,B 0,C 180,E1 -17636.346,E2 -17636.346} C_VEL
LIN {X 0,Y 275.435,Z 279.193,A -85,B 0,C 180,E1 -17638.538,E2 -17638.538} C_VEL
LIN {X 0,Y 275.502,Z 283.47,A -85,B 0,C 180,E1 -17640.731,E2 -17640.731} C_VEL
LIN {X 0,Y 275.912,Z 286.255,A -85,B 0,C 180,E1 -17642.92,E2 -17642.92} C_VEL
LIN {X 0,Y 276.419,Z 287.339,A -85,B 0,C 180,E1 -17644.375,E2 -17644.375} C_VEL
LIN {X 0,Y 277.146,Z 287.827,A -85,B 0,C 180,E1 -17645.822,E2 -17645.822} C_VEL
LIN {X 0,Y 277.693,Z 287.762,A -85,B 0,C 180,E1 -17647.27,E2 -17647.27} C_VEL
LIN {X 0,Y 278.869,Z 286.686,A -85,B 0,C 180,E1 -17649.17,E2 -17649.17} C_VEL
LIN {X 0,Y 279.574,Z 285.846,A -85,B 0,C 180,E1 -17650.135,E2 -17650.135} C_VEL
LIN {X 0,Y 281.62,Z 282.866,A -85,B 0,C 180,E1 -17652.247,E2 -17652.247} C_VEL
LIN {X 0,Y 282.538,Z 281.272,A -85,B 0,C 180,E1 -17653.086,E2 -17653.086} C_VEL
LIN {X 0,Y 282.819,Z 279.854,A -85,B 0,C 180,E1 -17653.843,E2 -17653.843} C_VEL
LIN {X 0,Y 280.544,Z 275.449,A -85,B 0,C 180,E1 -17656.407,E2 -17656.407} C_VEL
LIN {X 0,Y 280.996,Z 273.519,A -85,B 0,C 180,E1 -17657.109,E2 -17657.109} C_VEL
LIN {X 0,Y 284.437,Z 266.166,A -85,B 0,C 180,E1 -17659.083,E2 -17659.083} C_VEL
LIN {X 0,Y 285.478,Z 260.194,A -85,B 0,C 180,E1 -17660.687,E2 -17660.687} C_VEL
LIN {X 0,Y 285.716,Z 252.319,A -85,B 0,C 180,E1 -17662.746,E2 -17662.746} C_VEL
LIN {X 0,Y 285.066,Z 244.652,A -85,B 0,C 180,E1 -17664.779,E2 -17664.779} C_VEL
LIN {X 0,Y 283.473,Z 235.872,A -85,B 0,C 180,E1 -17667.24,E2 -17667.24} C_VEL
LIN {X 0,Y 281.888,Z 229.238,A -85,B 0,C 180,E1 -17669.233,E2 -17669.233} C_VEL
LIN {X 0,Y 280.752,Z 225.281,A -85,B 0,C 180,E1 -17670.555,E2 -17670.555} C_VEL
LIN {X 0,Y 279.004,Z 220.911,A -85,B 0,C 180,E1 -17672.363,E2 -17672.363} C_VEL
LIN {X 0,Y 278.728,Z 219.345,A -85,B 0,C 180,E1 -17672.903,E2 -17672.903} C_VEL
LIN {X 0,Y 279.219,Z 217.482,A -85,B 0,C 180,E1 -17676.344,E2 -17676.344} C_VEL
LIN {X 0,Y 279.329,Z 216.65,A -85,B 0,C 180,E1 -17678.977,E2 -17678.977} C_VEL
LIN {X 0,Y 279.438,Z 216.31,A -85,B 0,C 180,E1 -17681.014,E2 -17681.014} C_VEL
LIN {X 0,Y 279.684,Z 216.405,A -85,B 0,C 180,E1 -17684.716,E2 -17684.716} C_VEL
LIN {X 0,Y 279.903,Z 217.069,A -85,B 0,C 180,E1 -17687.315,E2 -17687.315} C_VEL
LIN {X 0,Y 280.253,Z 218.892,A -85,B 0,C 180,E1 -17691.023,E2 -17691.023} C_VEL
LIN {X 0,Y 280.456,Z 220.247,A -85,B 0,C 180,E1 -17692.914,E2 -17692.914} C_VEL
LIN {X 0,Y 282.005,Z 223.481,A -85,B 0,C 180,E1 -17694.153,E2 -17694.153} C_VEL
LIN {X 0,Y 284.25,Z 226.82,A -85,B 0,C 180,E1 -17695.585,E2 -17695.585} C_VEL
LIN {X 0,Y 287.116,Z 232.515,A -85,B 0,C 180,E1 -17697.415,E2 -17697.415} C_VEL
LIN {X 0,Y 288,Z 235.582,A -85,B 0,C 180,E1 -17698.152,E2 -17698.152} C_VEL
LIN {X 0,Y 289.171,Z 244.922,A -85,B 0,C 180,E1 -17699.961,E2 -17699.961} C_VEL
LIN {X 0,Y 289.536,Z 254.019,A -85,B 0,C 180,E1 -17701.641,E2 -17701.641} C_VEL
LIN {X 0,Y 289.055,Z 261.921,A -85,B 0,C 180,E1 -17703.072,E2 -17703.072} C_VEL
LIN {X 0,Y 288.235,Z 266.05,A -85,B 0,C 180,E1 -17703.77,E2 -17703.77} C_VEL
LIN {X 0,Y 285.087,Z 274.814,A -85,B 0,C 180,E1 -17705.221,E2 -17705.221} C_VEL
LIN {X 0,Y 281.274,Z 284.435,A -85,B 0,C 180,E1 -17707.212,E2 -17707.212} C_VEL
LIN {X 0,Y 277.952,Z 292.249,A -85,B 0,C 180,E1 -17709.266,E2 -17709.266} C_VEL
LIN {X 0,Y 275.173,Z 298.6,A -85,B 0,C 180,E1 -17711.38,E2 -17711.38} C_VEL
LIN {X 0,Y 273.063,Z 303.735,A -85,B 0,C 180,E1 -17713.552,E2 -17713.552} C_VEL
LIN {X 0,Y 271.092,Z 307.823,A -85,B 0,C 180,E1 -17715.74,E2 -17715.74} C_VEL
LIN {X 0,Y 269.77,Z 310.903,A -85,B 0,C 180,E1 -17717.968,E2 -17717.968} C_VEL
LIN {X 0,Y 269.154,Z 312.443,A -85,B 0,C 180,E1 -17719.466,E2 -17719.466} C_VEL
LIN {X 0,Y 268.412,Z 314.33,A -85,B 0,C 180,E1 -17722.475,E2 -17722.475} C_VEL
LIN {X 0,Y 268.342,Z 314.703,A -85,B 0,C 180,E1 -17724.409,E2 -17724.409} C_VEL
LIN {X 0,Y 268.345,Z 314.169,A -85,B 0,C 180,E1 -17726.995,E2 -17726.995} C_VEL
LIN {X 0,Y 268.687,Z 313.329,A -85,B 0,C 180,E1 -17728.499,E2 -17728.499} C_VEL
LIN {X 0,Y 268.825,Z 311.991,A -85,B 0,C 180,E1 -17729.998,E2 -17729.998} C_VEL
LIN {X 0,Y 268.843,Z 309.095,A -85,B 0,C 180,E1 -17732.245,E2 -17732.245} C_VEL
LIN {X 0,Y 268.836,Z 305.017,A -85,B 0,C 180,E1 -17734.496,E2 -17734.496} C_VEL
LIN {X 0,Y 268.915,Z 299.713,A -85,B 0,C 180,E1 -17736.724,E2 -17736.724} C_VEL
LIN {X 0,Y 269.08,Z 292.659,A -85,B 0,C 180,E1 -17739.014,E2 -17739.014} C_VEL
LIN {X 0,Y 269.384,Z 285.439,A -85,B 0,C 180,E1 -17740.9,E2 -17740.9} C_VEL
LIN {X 0,Y 269.902,Z 276.567,A -85,B 0,C 180,E1 -17742.785,E2 -17742.785} C_VEL
LIN {X 0,Y 270.494,Z 267.891,A -85,B 0,C 180,E1 -17744.287,E2 -17744.287} C_VEL
LIN {X 0,Y 271.244,Z 257.275,A -85,B 0,C 180,E1 -17745.784,E2 -17745.784} C_VEL
LIN {X 0,Y 271.807,Z 247.096,A -85,B 0,C 180,E1 -17746.923,E2 -17746.923} C_VEL
LIN {X 0,Y 270.589,Z 233.605,A -85,B 0,C 180,E1 -17748.069,E2 -17748.069} C_VEL
LIN {X 0,Y 270.008,Z 221.579,A -85,B 0,C 180,E1 -17748.788,E2 -17748.788} C_VEL
LIN {X 0,Y 270.022,Z 219.996,A -85,B 0,C 180,E1 -17748.885,E2 -17748.885} C_VEL
LIN {X 0,Y 271.771,Z 207.544,A -85,B 0,C 180,E1 -17754.438,E2 -17754.438} C_VEL
LIN {X 0,Y 273.454,Z 198.777,A -85,B 0,C 180,E1 -17758.365,E2 -17758.365} C_VEL
LIN {X 0,Y 273.639,Z 196.932,A -85,B 0,C 180,E1 -17759.205,E2 -17759.205} C_VEL
LIN {X 0,Y 272.641,Z 191.649,A -85,B 0,C 180,E1 -17761.716,E2 -17761.716} C_VEL
LIN {X 0,Y 270.856,Z 182.036,A -85,B 0,C 180,E1 -17766.45,E2 -17766.45} C_VEL
LIN {X 0,Y 270.27,Z 178.825,A -85,B 0,C 180,E1 -17768.136,E2 -17768.136} C_VEL
LIN {X 0,Y 270.179,Z 178.832,A -85,B 0,C 180,E1 -17772.553,E2 -17772.553} C_VEL
LIN {X 0,Y 270.204,Z 178.825,A -85,B 0,C 180,E1 -17776.738,E2 -17776.738} C_VEL
LIN {X 0,Y 270.237,Z 178.82,A -85,B 0,C 180,E1 -17779.445,E2 -17779.445} C_VEL
LIN {X 0,Y 270.247,Z 178.82,A -85,B 0,C 180,E1 -17783.719,E2 -17783.719} C_VEL
LIN {X 0,Y 270.193,Z 178.825,A -85,B 0,C 180,E1 -17786.891,E2 -17786.891} C_VEL
LIN {X 0,Y 270.186,Z 178.829,A -85,B 0,C 180,E1 -17790.381,E2 -17790.381} C_VEL
LIN {X 0,Y 270.25,Z 178.822,A -85,B 0,C 180,E1 -17793.762,E2 -17793.762} C_VEL
LIN {X 0,Y 270.198,Z 178.826,A -85,B 0,C 180,E1 -17797.035,E2 -17797.035} C_VEL
LIN {X 0,Y 270.289,Z 178.815,A -85,B 0,C 180,E1 -17800.243,E2 -17800.243} C_VEL
LIN {X 0,Y 270.39,Z 178.802,A -85,B 0,C 180,E1 -17804.934,E2 -17804.934} C_VEL
LIN {X 0,Y 270.429,Z 178.799,A -85,B 0,C 180,E1 -17809.518,E2 -17809.518} C_VEL
LIN {X 0,Y 270.595,Z 178.775,A -85,B 0,C 180,E1 -17812.538,E2 -17812.538} C_VEL
LIN {X 0,Y 270.777,Z 178.754,A -85,B 0,C 180,E1 -17818.513,E2 -17818.513} C_VEL
LIN {X 0,Y 270.772,Z 178.755,A -85,B 0,C 180,E1 -17821.487,E2 -17821.487} C_VEL
LIN {X 0,Y 270.597,Z 178.775,A -85,B 0,C 180,E1 -17827.461,E2 -17827.461} C_VEL
LIN {X 0,Y 270.429,Z 178.799,A -85,B 0,C 180,E1 -17830.481,E2 -17830.481} C_VEL
LIN {X 0,Y 270.39,Z 178.802,A -85,B 0,C 180,E1 -17835.065,E2 -17835.065} C_VEL
LIN {X 0,Y 270.29,Z 178.815,A -85,B 0,C 180,E1 -17839.756,E2 -17839.756} C_VEL
LIN {X 0,Y 270.214,Z 178.824,A -85,B 0,C 180,E1 -17844.591,E2 -17844.591} C_VEL
LIN {X 0,Y 270.191,Z 178.829,A -85,B 0,C 180,E1 -17847.918,E2 -17847.918} C_VEL
LIN {X 0,Y 270.161,Z 178.831,A -85,B 0,C 180,E1 -17851.351,E2 -17851.351} C_VEL
LIN {X 0,Y 270.203,Z 178.823,A -85,B 0,C 180,E1 -17854.905,E2 -17854.905} C_VEL
LIN {X 0,Y 270.212,Z 178.824,A -85,B 0,C 180,E1 -17858.719,E2 -17858.719} C_VEL
LIN {X 0,Y 270.182,Z 178.826,A -85,B 0,C 180,E1 -17862.556,E2 -17862.556} C_VEL
LIN {X 0,Y 270.163,Z 178.83,A -85,B 0,C 180,E1 -17866.752,E2 -17866.752} C_VEL
LIN {X 0,Y 270.189,Z 178.829,A -85,B 0,C 180,E1 -17871.292,E2 -17871.292} C_VEL
LIN {X 0,Y 270.195,Z 178.83,A -85,B 0,C 180,E1 -17875.097,E2 -17875.097} C_VEL
LIN {X 0,Y 270.194,Z 178.828,A -85,B 0,C 180,E1 -17879.133,E2 -17879.133} C_VEL
LIN {X 0,Y 270.26,Z 178.818,A -85,B 0,C 180,E1 -17882.148,E2 -17882.148} C_VEL
LIN {X 0,Y 270.273,Z 178.816,A -85,B 0,C 180,E1 -17885.522,E2 -17885.522} C_VEL
LIN {X 0,Y 270.299,Z 178.814,A -85,B 0,C 180,E1 -17890.247,E2 -17890.247} C_VEL
LIN {X 0,Y 270.401,Z 178.801,A -85,B 0,C 180,E1 -17894.938,E2 -17894.938} C_VEL
LIN {X 0,Y 270.441,Z 178.795,A -85,B 0,C 180,E1 -17899.521,E2 -17899.521} C_VEL
LIN {X 0,Y 270.612,Z 178.776,A -85,B 0,C 180,E1 -17902.541,E2 -17902.541} C_VEL
LIN {X 0,Y 270.78,Z 178.754,A -85,B 0,C 180,E1 -17908.515,E2 -17908.515} C_VEL
LIN {X 0,Y 270.779,Z 178.755,A -85,B 0,C 180,E1 -17911.49,E2 -17911.49} C_VEL
LIN {X 0,Y 270.614,Z 178.776,A -85,B 0,C 180,E1 -17917.463,E2 -17917.463} C_VEL
LIN {X 0,Y 270.445,Z 178.795,A -85,B 0,C 180,E1 -17920.483,E2 -17920.483} C_VEL
LIN {X 0,Y 270.407,Z 178.8,A -85,B 0,C 180,E1 -17925.067,E2 -17925.067} C_VEL
LIN {X 0,Y 270.294,Z 178.814,A -85,B 0,C 180,E1 -17929.758,E2 -17929.758} C_VEL
LIN {X 0,Y 270.181,Z 178.828,A -85,B 0,C 180,E1 -17934.597,E2 -17934.597} C_VEL
LIN {X 0,Y 270.201,Z 178.825,A -85,B 0,C 180,E1 -17937.919,E2 -17937.919} C_VEL
LIN {X 0,Y 270.178,Z 178.829,A -85,B 0,C 180,E1 -17941.351,E2 -17941.351} C_VEL
LIN {X 0,Y 270.204,Z 178.829,A -85,B 0,C 180,E1 -17944.907,E2 -17944.907} C_VEL
LIN {X 0,Y 270.203,Z 178.828,A -85,B 0,C 180,E1 -17948.712,E2 -17948.712} C_VEL
LIN {X 0,Y 270.154,Z 178.832,A -85,B 0,C 180,E1 -17953.246,E2 -17953.246} C_VEL
LIN {X 0,Y 270.185,Z 178.825,A -85,B 0,C 180,E1 -17957.444,E2 -17957.444} C_VEL
LIN {X 0,Y 270.214,Z 178.824,A -85,B 0,C 180,E1 -17961.375,E2 -17961.375} C_VEL
LIN {X 0,Y 270.369,Z 178.977,A -85,B 0,C 180,E1 -17964.892,E2 -17964.892} C_VEL
LIN {X 0,Y 271.25,Z 183.689,A -85,B 0,C 180,E1 -17967.918,E2 -17967.918} C_VEL
LIN {X 0,Y 271.202,Z 187.898,A -85,B 0,C 180,E1 -17970.503,E2 -17970.503} C_VEL
LIN {X 0,Y 270.38,Z 194.744,A -85,B 0,C 180,E1 -17974.603,E2 -17974.603} C_VEL
LIN {X 0,Y 269.75,Z 201.516,A -85,B 0,C 180,E1 -17978.608,E2 -17978.608} C_VEL
LIN {X 0,Y 269.231,Z 208.214,A -85,B 0,C 180,E1 -17982.531,E2 -17982.531} C_VEL
LIN {X 0,Y 268.84,Z 217.007,A -85,B 0,C 180,E1 -17987.497,E2 -17987.497} C_VEL
LIN {X 0,Y 269.433,Z 228.109,A -85,B 0,C 180,E1 -17988.432,E2 -17988.432} C_VEL
LIN {X 0,Y 270.198,Z 237.983,A -85,B 0,C 180,E1 -17989.51,E2 -17989.51} C_VEL
LIN {X 0,Y 269.697,Z 248.689,A -85,B 0,C 180,E1 -17991.005,E2 -17991.005} C_VEL
LIN {X 0,Y 269.162,Z 258.666,A -85,B 0,C 180,E1 -17992.787,E2 -17992.787} C_VEL
LIN {X 0,Y 268.857,Z 267.237,A -85,B 0,C 180,E1 -17994.751,E2 -17994.751} C_VEL
LIN {X 0,Y 268.557,Z 273.668,A -85,B 0,C 180,E1 -17996.625,E2 -17996.625} C_VEL
LIN {X 0,Y 268.358,Z 278.722,A -85,B 0,C 180,E1 -17998.499,E2 -17998.499} C_VEL
LIN {X 0,Y 268.419,Z 283.251,A -85,B 0,C 180,E1 -18000.75,E2 -18000.75} C_VEL
LIN {X 0,Y 268.835,Z 286.312,A -85,B 0,C 180,E1 -18002.997,E2 -18002.997} C_VEL
LIN {X 0,Y 269.352,Z 287.593,A -85,B 0,C 180,E1 -18004.49,E2 -18004.49} C_VEL
LIN {X 0,Y 270.093,Z 288.263,A -85,B 0,C 180,E1 -18005.974,E2 -18005.974} C_VEL
LIN {X 0,Y 270.677,Z 288.359,A -85,B 0,C 180,E1 -18007.459,E2 -18007.459} C_VEL
LIN {X 0,Y 271.597,Z 287.89,A -85,B 0,C 180,E1 -18008.932,E2 -18008.932} C_VEL
LIN {X 0,Y 272.671,Z 286.868,A -85,B 0,C 180,E1 -18010.395,E2 -18010.395} C_VEL
LIN {X 0,Y 274.803,Z 284.196,A -85,B 0,C 180,E1 -18012.556,E2 -18012.556} C_VEL
LIN {X 0,Y 277.387,Z 280.165,A -85,B 0,C 180,E1 -18014.677,E2 -18014.677} C_VEL
LIN {X 0,Y 280.43,Z 274.654,A -85,B 0,C 180,E1 -18016.751,E2 -18016.751} C_VEL
LIN {X 0,Y 280.996,Z 273.519,A -85,B 0,C 180,E1 -18017.109,E2 -18017.109} C_VEL
LIN {X 0,Y 281.964,Z 270.44,A -85,B 0,C 180,E1 -18018.115,E2 -18018.115} C_VEL
LIN {X 0,Y 281.887,Z 267.585,A -85,B 0,C 180,E1 -18019.178,E2 -18019.178} C_VEL
LIN {X 0,Y 280.097,Z 259.925,A -85,B 0,C 180,E1 -18022.059,E2 -18022.059} C_VEL
LIN {X 0,Y 280.022,Z 257.665,A -85,B 0,C 180,E1 -18022.746,E2 -18022.746} C_VEL
LIN {X 0,Y 279.873,Z 248.82,A -85,B 0,C 180,E1 -18025.271,E2 -18025.271} C_VEL
LIN {X 0,Y 278.929,Z 241.137,A -85,B 0,C 180,E1 -18027.573,E2 -18027.573} C_VEL
LIN {X 0,Y 277.814,Z 234.667,A -85,B 0,C 180,E1 -18029.649,E2 -18029.649} C_VEL
LIN {X 0,Y 276.919,Z 230.84,A -85,B 0,C 180,E1 -18031.025,E2 -18031.025} C_VEL
LIN {X 0,Y 275.199,Z 225.101,A -85,B 0,C 180,E1 -18033.509,E2 -18033.509} C_VEL
LIN {X 0,Y 272.619,Z 219.62,A -85,B 0,C 180,E1 -18037.522,E2 -18037.522} C_VEL
LIN {X 0,Y 272.749,Z 219.035,A -85,B 0,C 180,E1 -18040.105,E2 -18040.105} C_VEL
LIN {X 0,Y 272.995,Z 218.98,A -85,B 0,C 180,E1 -18043.874,E2 -18043.874} C_VEL
LIN {X 0,Y 273.228,Z 219.358,A -85,B 0,C 180,E1 -18046.073,E2 -18046.073} C_VEL
LIN {X 0,Y 273.37,Z 220.104,A -85,B 0,C 180,E1 -18048.207,E2 -18048.207} C_VEL
LIN {X 0,Y 276.669,Z 225.592,A -85,B 0,C 180,E1 -18051.95,E2 -18051.95} C_VEL
LIN {X 0,Y 277.428,Z 226.525,A -85,B 0,C 180,E1 -18052.554,E2 -18052.554} C_VEL
LIN {X 0,Y 279.394,Z 230.562,A -85,B 0,C 180,E1 -18054.274,E2 -18054.274} C_VEL
LIN {X 0,Y 281.146,Z 233.79,A -85,B 0,C 180,E1 -18055.581,E2 -18055.581} C_VEL
LIN {X 0,Y 282.888,Z 237.501,A -85,B 0,C 180,E1 -18056.866,E2 -18056.866} C_VEL
LIN {X 0,Y 283.642,Z 241.221,A -85,B 0,C 180,E1 -18057.767,E2 -18057.767} C_VEL
LIN {X 0,Y 284.2,Z 251.87,A -85,B 0,C 180,E1 -18059.942,E2 -18059.942} C_VEL
LIN {X 0,Y 283.701,Z 261.933,A -85,B 0,C 180,E1 -18061.92,E2 -18061.92} C_VEL
LIN {X 0,Y 283.069,Z 265.806,A -85,B 0,C 180,E1 -18062.655,E2 -18062.655} C_VEL
LIN {X 0,Y 279.561,Z 275.246,A -85,B 0,C 180,E1 -18064.298,E2 -18064.298} C_VEL
LIN {X 0,Y 275.539,Z 284.657,A -85,B 0,C 180,E1 -18066.312,E2 -18066.312} C_VEL
LIN {X 0,Y 271.424,Z 293.422,A -85,B 0,C 180,E1 -18068.744,E2 -18068.744} C_VEL
LIN {X 0,Y 269.394,Z 297.551,A -85,B 0,C 180,E1 -18070.173,E2 -18070.173} C_VEL
LIN {X 0,Y 267.03,Z 302.754,A -85,B 0,C 180,E1 -18072.38,E2 -18072.38} C_VEL
LIN {X 0,Y 264.852,Z 306.912,A -85,B 0,C 180,E1 -18074.61,E2 -18074.61} C_VEL
LIN {X 0,Y 263.644,Z 309.148,A -85,B 0,C 180,E1 -18076.116,E2 -18076.116} C_VEL
LIN {X 0,Y 262.135,Z 312.323,A -85,B 0,C 180,E1 -18079.181,E2 -18079.181} C_VEL
LIN {X 0,Y 261.673,Z 313.349,A -85,B 0,C 180,E1 -18080.724,E2 -18080.724} C_VEL
LIN {X 0,Y 261.229,Z 314.173,A -85,B 0,C 180,E1 -18083.82,E2 -18083.82} C_VEL
LIN {X 0,Y 261.298,Z 314.022,A -85,B 0,C 180,E1 -18085.369,E2 -18085.369} C_VEL
LIN {X 0,Y 261.283,Z 313.432,A -85,B 0,C 180,E1 -18086.914,E2 -18086.914} C_VEL
LIN {X 0,Y 261.642,Z 312.448,A -85,B 0,C 180,E1 -18088.458,E2 -18088.458} C_VEL
LIN {X 0,Y 261.808,Z 311.027,A -85,B 0,C 180,E1 -18089.998,E2 -18089.998} C_VEL
LIN {X 0,Y 261.828,Z 307.934,A -85,B 0,C 180,E1 -18092.305,E2 -18092.305} C_VEL
LIN {X 0,Y 261.833,Z 303.624,A -85,B 0,C 180,E1 -18094.616,E2 -18094.616} C_VEL
LIN {X 0,Y 261.954,Z 297.006,A -85,B 0,C 180,E1 -18097.279,E2 -18097.279} C_VEL
LIN {X 0,Y 262.126,Z 289.276,A -85,B 0,C 180,E1 -18099.644,E2 -18099.644} C_VEL
LIN {X 0,Y 262.549,Z 281.426,A -85,B 0,C 180,E1 -18101.579,E2 -18101.579} C_VEL
LIN {X 0,Y 263.238,Z 271.733,A -85,B 0,C 180,E1 -18103.507,E2 -18103.507} C_VEL
LIN {X 0,Y 263.892,Z 260.768,A -85,B 0,C 180,E1 -18105.245,E2 -18105.245} C_VEL
LIN {X 0,Y 264.693,Z 248.882,A -85,B 0,C 180,E1 -18106.706,E2 -18106.706} C_VEL
LIN {X 0,Y 263.899,Z 238.217,A -85,B 0,C 180,E1 -18107.72,E2 -18107.72} C_VEL
LIN {X 0,Y 263.049,Z 225.836,A -85,B 0,C 180,E1 -18108.596,E2 -18108.596} C_VEL
LIN {X 0,Y 262.922,Z 220.014,A -85,B 0,C 180,E1 -18108.909,E2 -18108.909} C_VEL
LIN {X 0,Y 264.601,Z 208.309,A -85,B 0,C 180,E1 -18114.308,E2 -18114.308} C_VEL
LIN {X 0,Y 266.338,Z 199.54,A -85,B 0,C 180,E1 -18118.355,E2 -18118.355} C_VEL
LIN {X 0,Y 266.383,Z 195.911,A -85,B 0,C 180,E1 -18120.081,E2 -18120.081} C_VEL
LIN {X 0,Y 264.32,Z 185.816,A -85,B 0,C 180,E1 -18125.114,E2 -18125.114} C_VEL
LIN {X 0,Y 263.212,Z 179.702,A -85,B 0,C 180,E1 -18128.363,E2 -18128.363} C_VEL
LIN {X 0,Y 263.124,Z 179.707,A -85,B 0,C 180,E1 -18131.89,E2 -18131.89} C_VEL
LIN {X 0,Y 263.138,Z 179.706,A -85,B 0,C 180,E1 -18136.143,E2 -18136.143} C_VEL
LIN {X 0,Y 263.151,Z 179.706,A -85,B 0,C 180,E1 -18140.136,E2 -18140.136} C_VEL
LIN {X 0,Y 263.18,Z 179.703,A -85,B 0,C 180,E1 -18144.021,E2 -18144.021} C_VEL
LIN {X 0,Y 263.123,Z 179.708,A -85,B 0,C 180,E1 -18147.71,E2 -18147.71} C_VEL
LIN {X 0,Y 263.185,Z 179.702,A -85,B 0,C 180,E1 -18151.783,E2 -18151.783} C_VEL
LIN {X 0,Y 263.189,Z 179.698,A -85,B 0,C 180,E1 -18155.211,E2 -18155.211} C_VEL
LIN {X 0,Y 263.25,Z 179.695,A -85,B 0,C 180,E1 -18159.692,E2 -18159.692} C_VEL
LIN {X 0,Y 263.338,Z 179.679,A -85,B 0,C 180,E1 -18164.521,E2 -18164.521} C_VEL
LIN {X 0,Y 263.361,Z 179.681,A -85,B 0,C 180,E1 -18169.234,E2 -18169.234} C_VEL
LIN {X 0,Y 263.557,Z 179.652,A -85,B 0,C 180,E1 -18172.338,E2 -18172.338} C_VEL
LIN {X 0,Y 263.742,Z 179.63,A -85,B 0,C 180,E1 -18178.473,E2 -18178.473} C_VEL
LIN {X 0,Y 263.737,Z 179.631,A -85,B 0,C 180,E1 -18181.527,E2 -18181.527} C_VEL
LIN {X 0,Y 263.559,Z 179.651,A -85,B 0,C 180,E1 -18187.662,E2 -18187.662} C_VEL
LIN {X 0,Y 263.361,Z 179.681,A -85,B 0,C 180,E1 -18190.766,E2 -18190.766} C_VEL
LIN {X 0,Y 263.338,Z 179.679,A -85,B 0,C 180,E1 -18195.479,E2 -18195.479} C_VEL
LIN {X 0,Y 263.251,Z 179.695,A -85,B 0,C 180,E1 -18200.308,E2 -18200.308} C_VEL
LIN {X 0,Y 263.158,Z 179.701,A -85,B 0,C 180,E1 -18205.296,E2 -18205.296} C_VEL
LIN {X 0,Y 263.124,Z 179.707,A -85,B 0,C 180,E1 -18208.736,E2 -18208.736} C_VEL
LIN {X 0,Y 263.117,Z 179.709,A -85,B 0,C 180,E1 -18212.29,E2 -18212.29} C_VEL
LIN {X 0,Y 263.177,Z 179.703,A -85,B 0,C 180,E1 -18215.98,E2 -18215.98} C_VEL
LIN {X 0,Y 263.113,Z 179.711,A -85,B 0,C 180,E1 -18219.871,E2 -18219.871} C_VEL
LIN {X 0,Y 263.124,Z 179.707,A -85,B 0,C 180,E1 -18223.984,E2 -18223.984} C_VEL
LIN {X 0,Y 263.116,Z 179.708,A -85,B 0,C 180,E1 -18228.409,E2 -18228.409} C_VEL
LIN {X 0,Y 263.175,Z 179.704,A -85,B 0,C 180,E1 -18233.239,E2 -18233.239} C_VEL
LIN {X 0,Y 263.127,Z 179.706,A -85,B 0,C 180,E1 -18237.714,E2 -18237.714} C_VEL
LIN {X 0,Y 263.196,Z 179.697,A -85,B 0,C 180,E1 -18241.785,E2 -18241.785} C_VEL
LIN {X 0,Y 263.222,Z 179.696,A -85,B 0,C 180,E1 -18245.203,E2 -18245.203} C_VEL
LIN {X 0,Y 263.261,Z 179.689,A -85,B 0,C 180,E1 -18249.696,E2 -18249.696} C_VEL
LIN {X 0,Y 263.349,Z 179.683,A -85,B 0,C 180,E1 -18254.525,E2 -18254.525} C_VEL
LIN {X 0,Y 263.373,Z 179.675,A -85,B 0,C 180,E1 -18259.237,E2 -18259.237} C_VEL
LIN {X 0,Y 263.573,Z 179.654,A -85,B 0,C 180,E1 -18262.341,E2 -18262.341} C_VEL
LIN {X 0,Y 263.746,Z 179.631,A -85,B 0,C 180,E1 -18268.475,E2 -18268.475} C_VEL
LIN {X 0,Y 263.745,Z 179.631,A -85,B 0,C 180,E1 -18271.529,E2 -18271.529} C_VEL
LIN {X 0,Y 263.576,Z 179.654,A -85,B 0,C 180,E1 -18277.664,E2 -18277.664} C_VEL
LIN {X 0,Y 263.377,Z 179.675,A -85,B 0,C 180,E1 -18280.768,E2 -18280.768} C_VEL
LIN {X 0,Y 263.355,Z 179.682,A -85,B 0,C 180,E1 -18285.48,E2 -18285.48} C_VEL
LIN {X 0,Y 263.254,Z 179.689,A -85,B 0,C 180,E1 -18290.31,E2 -18290.31} C_VEL
LIN {X 0,Y 263.13,Z 179.71,A -85,B 0,C 180,E1 -18295.302,E2 -18295.302} C_VEL
LIN {X 0,Y 263.137,Z 179.707,A -85,B 0,C 180,E1 -18298.737,E2 -18298.737} C_VEL
LIN {X 0,Y 263.133,Z 179.706,A -85,B 0,C 180,E1 -18302.291,E2 -18302.291} C_VEL
LIN {X 0,Y 263.184,Z 179.703,A -85,B 0,C 180,E1 -18306.763,E2 -18306.763} C_VEL
LIN {X 0,Y 263.097,Z 179.709,A -85,B 0,C 180,E1 -18309.877,E2 -18309.877} C_VEL
LIN {X 0,Y 263.104,Z 179.71,A -85,B 0,C 180,E1 -18313.991,E2 -18313.991} C_VEL
LIN {X 0,Y 263.135,Z 179.706,A -85,B 0,C 180,E1 -18318.109,E2 -18318.109} C_VEL
LIN {X 0,Y 263.177,Z 179.704,A -85,B 0,C 180,E1 -18322.106,E2 -18322.106} C_VEL
LIN {X 0,Y 263.319,Z 179.69,A -85,B 0,C 180,E1 -18324.716,E2 -18324.716} C_VEL
LIN {X 0,Y 264.251,Z 185.191,A -85,B 0,C 180,E1 -18328.331,E2 -18328.331} C_VEL
LIN {X 0,Y 264.124,Z 188.67,A -85,B 0,C 180,E1 -18330.511,E2 -18330.511} C_VEL
LIN {X 0,Y 263.264,Z 195.542,A -85,B 0,C 180,E1 -18334.714,E2 -18334.714} C_VEL
LIN {X 0,Y 262.627,Z 202.331,A -85,B 0,C 180,E1 -18338.823,E2 -18338.823} C_VEL
LIN {X 0,Y 262.074,Z 209.05,A -85,B 0,C 180,E1 -18342.843,E2 -18342.843} C_VEL
LIN {X 0,Y 261.756,Z 216.816,A -85,B 0,C 180,E1 -18347.449,E2 -18347.449} C_VEL
LIN {X 0,Y 262.379,Z 228.809,A -85,B 0,C 180,E1 -18348.509,E2 -18348.509} C_VEL
LIN {X 0,Y 263.085,Z 238.531,A -85,B 0,C 180,E1 -18349.612,E2 -18349.612} C_VEL
LIN {X 0,Y 262.578,Z 249.165,A -85,B 0,C 180,E1 -18351.147,E2 -18351.147} C_VEL
LIN {X 0,Y 262.07,Z 258.536,A -85,B 0,C 180,E1 -18352.87,E2 -18352.87} C_VEL
LIN {X 0,Y 261.809,Z 266.121,A -85,B 0,C 180,E1 -18354.609,E2 -18354.609} C_VEL
LIN {X 0,Y 261.499,Z 272.836,A -85,B 0,C 180,E1 -18356.533,E2 -18356.533} C_VEL
LIN {X 0,Y 261.284,Z 278.157,A -85,B 0,C 180,E1 -18358.459,E2 -18358.459} C_VEL
LIN {X 0,Y 261.337,Z 282.986,A -85,B 0,C 180,E1 -18360.771,E2 -18360.771} C_VEL
LIN {X 0,Y 261.761,Z 286.31,A -85,B 0,C 180,E1 -18363.078,E2 -18363.078} C_VEL
LIN {X 0,Y 262.287,Z 287.753,A -85,B 0,C 180,E1 -18364.611,E2 -18364.611} C_VEL
LIN {X 0,Y 263.038,Z 288.62,A -85,B 0,C 180,E1 -18366.135,E2 -18366.135} C_VEL
LIN {X 0,Y 263.663,Z 288.933,A -85,B 0,C 180,E1 -18367.659,E2 -18367.659} C_VEL
LIN {X 0,Y 264.641,Z 288.643,A -85,B 0,C 180,E1 -18369.169,E2 -18369.169} C_VEL
LIN {X 0,Y 265.772,Z 287.811,A -85,B 0,C 180,E1 -18370.667,E2 -18370.667} C_VEL
LIN {X 0,Y 267.281,Z 286.406,A -85,B 0,C 180,E1 -18372.143,E2 -18372.143} C_VEL
LIN {X 0,Y 269.769,Z 283.209,A -85,B 0,C 180,E1 -18374.329,E2 -18374.329} C_VEL
LIN {X 0,Y 272.799,Z 278.603,A -85,B 0,C 180,E1 -18376.463,E2 -18376.463} C_VEL
LIN {X 0,Y 275.626,Z 273.63,A -85,B 0,C 180,E1 -18378.201,E2 -18378.201} C_VEL
LIN {X 0,Y 278.623,Z 267.494,A -85,B 0,C 180,E1 -18379.909,E2 -18379.909} C_VEL
LIN {X 0,Y 279.719,Z 261.614,A -85,B 0,C 180,E1 -18381.618,E2 -18381.618} C_VEL
LIN {X 0,Y 280.022,Z 257.665,A -85,B 0,C 180,E1 -18382.746,E2 -18382.746} C_VEL
LIN {X 0,Y 279.626,Z 254.574,A -85,B 0,C 180,E1 -18383.77,E2 -18383.77} C_VEL
LIN {X 0,Y 278.436,Z 252.088,A -85,B 0,C 180,E1 -18384.85,E2 -18384.85} C_VEL
LIN {X 0,Y 274.527,Z 246.172,A -85,B 0,C 180,E1 -18387.832,E2 -18387.832} C_VEL
LIN {X 0,Y 274.014,Z 244.329,A -85,B 0,C 180,E1 -18388.569,E2 -18388.569} C_VEL
LIN {X 0,Y 273.272,Z 238.855,A -85,B 0,C 180,E1 -18390.539,E2 -18390.539} C_VEL
LIN {X 0,Y 272.768,Z 235.722,A -85,B 0,C 180,E1 -18391.757,E2 -18391.757} C_VEL
LIN {X 0,Y 271.577,Z 230.828,A -85,B 0,C 180,E1 -18394.092,E2 -18394.092} C_VEL
LIN {X 0,Y 270.114,Z 227.257,A -85,B 0,C 180,E1 -18396.758,E2 -18396.758} C_VEL
LIN {X 0,Y 269.31,Z 225.539,A -85,B 0,C 180,E1 -18398.779,E2 -18398.779} C_VEL
LIN {X 0,Y 268.733,Z 224.809,A -85,B 0,C 180,E1 -18400.83,E2 -18400.83} C_VEL
LIN {X 0,Y 268.681,Z 224.608,A -85,B 0,C 180,E1 -18402.909,E2 -18402.909} C_VEL
LIN {X 0,Y 269.186,Z 225.111,A -85,B 0,C 180,E1 -18405.174,E2 -18405.174} C_VEL
LIN {X 0,Y 270.354,Z 226.312,A -85,B 0,C 180,E1 -18407.475,E2 -18407.475} C_VEL
LIN {X 0,Y 271.726,Z 229.093,A -85,B 0,C 180,E1 -18409.711,E2 -18409.711} C_VEL
LIN {X 0,Y 273.903,Z 232.294,A -85,B 0,C 180,E1 -18411.987,E2 -18411.987} C_VEL
LIN {X 0,Y 277.013,Z 238.769,A -85,B 0,C 180,E1 -18414.961,E2 -18414.961} C_VEL
LIN {X 0,Y 278.577,Z 242.57,A -85,B 0,C 180,E1 -18416.36,E2 -18416.36} C_VEL
LIN {X 0,Y 279.026,Z 246.64,A -85,B 0,C 180,E1 -18417.374,E2 -18417.374} C_VEL
LIN {X 0,Y 278.885,Z 257.502,A -85,B 0,C 180,E1 -18419.732,E2 -18419.732} C_VEL
LIN {X 0,Y 277.667,Z 266.77,A -85,B 0,C 180,E1 -18421.666,E2 -18421.666} C_VEL
LIN {X 0,Y 275.645,Z 272.339,A -85,B 0,C 180,E1 -18422.679,E2 -18422.679} C_VEL
LIN {X 0,Y 271.235,Z 282.112,A -85,B 0,C 180,E1 -18424.687,E2 -18424.687} C_VEL
LIN {X 0,Y 267.278,Z 290.087,A -85,B 0,C 180,E1 -18426.768,E2 -18426.768} C_VEL
LIN {X 0,Y 263.317,Z 297.375,A -85,B 0,C 180,E1 -18429.214,E2 -18429.214} C_VEL
LIN {X 0,Y 260.3,Z 303.373,A -85,B 0,C 180,E1 -18431.909,E2 -18431.909} C_VEL
LIN {X 0,Y 257.365,Z 308.322,A -85,B 0,C 180,E1 -18434.962,E2 -18434.962} C_VEL
LIN {X 0,Y 255.823,Z 310.937,A -85,B 0,C 180,E1 -18437.302,E2 -18437.302} C_VEL
LIN {X 0,Y 255.132,Z 312.196,A -85,B 0,C 180,E1 -18438.88,E2 -18438.88} C_VEL
LIN {X 0,Y 254.302,Z 313.533,A -85,B 0,C 180,E1 -18442.055,E2 -18442.055} C_VEL
LIN {X 0,Y 254.211,Z 313.536,A -85,B 0,C 180,E1 -18444.426,E2 -18444.426} C_VEL
LIN {X 0,Y 254.23,Z 312.62,A -85,B 0,C 180,E1 -18446.828,E2 -18446.828} C_VEL
LIN {X 0,Y 254.597,Z 311.548,A -85,B 0,C 180,E1 -18448.416,E2 -18448.416} C_VEL
LIN {X 0,Y 254.782,Z 309.003,A -85,B 0,C 180,E1 -18450.788,E2 -18450.788} C_VEL
LIN {X 0,Y 254.783,Z 305.289,A -85,B 0,C 180,E1 -18453.16,E2 -18453.16} C_VEL
LIN {X 0,Y 254.867,Z 300.313,A -85,B 0,C 180,E1 -18455.536,E2 -18455.536} C_VEL
LIN {X 0,Y 254.967,Z 293.853,A -85,B 0,C 180,E1 -18457.919,E2 -18457.919} C_VEL
LIN {X 0,Y 255.131,Z 287.104,A -85,B 0,C 180,E1 -18459.911,E2 -18459.911} C_VEL
LIN {X 0,Y 255.587,Z 278.841,A -85,B 0,C 180,E1 -18461.899,E2 -18461.899} C_VEL
LIN {X 0,Y 256.275,Z 268.664,A -85,B 0,C 180,E1 -18463.881,E2 -18463.881} C_VEL
LIN {X 0,Y 257.061,Z 256.981,A -85,B 0,C 180,E1 -18465.66,E2 -18465.66} C_VEL
LIN {X 0,Y 257.622,Z 248.072,A -85,B 0,C 180,E1 -18466.74,E2 -18466.74} C_VEL
LIN {X 0,Y 256.624,Z 236.524,A -85,B 0,C 180,E1 -18467.839,E2 -18467.839} C_VEL
LIN {X 0,Y 255.845,Z 223.956,A -85,B 0,C 180,E1 -18468.724,E2 -18468.724} C_VEL
LIN {X 0,Y 255.833,Z 220.031,A -85,B 0,C 180,E1 -18468.933,E2 -18468.933} C_VEL
LIN {X 0,Y 257.424,Z 209.026,A -85,B 0,C 180,E1 -18474.172,E2 -18474.172} C_VEL
LIN {X 0,Y 259.189,Z 200.285,A -85,B 0,C 180,E1 -18478.325,E2 -18478.325} C_VEL
LIN {X 0,Y 259.383,Z 197.081,A -85,B 0,C 180,E1 -18479.883,E2 -18479.883} C_VEL
LIN {X 0,Y 257.356,Z 187.151,A -85,B 0,C 180,E1 -18484.99,E2 -18484.99} C_VEL
LIN {X 0,Y 256.15,Z 180.579,A -85,B 0,C 180,E1 -18488.551,E2 -18488.551} C_VEL
LIN {X 0,Y 256.065,Z 180.586,A -85,B 0,C 180,E1 -18493.322,E2 -18493.322} C_VEL
LIN {X 0,Y 256.116,Z 180.578,A -85,B 0,C 180,E1 -18497.803,E2 -18497.803} C_VEL
LIN {X 0,Y 256.1,Z 180.583,A -85,B 0,C 180,E1 -18500.863,E2 -18500.863} C_VEL
LIN {X 0,Y 256.112,Z 180.579,A -85,B 0,C 180,E1 -18504.812,E2 -18504.812} C_VEL
LIN {X 0,Y 256.082,Z 180.585,A -85,B 0,C 180,E1 -18508.571,E2 -18508.571} C_VEL
LIN {X 0,Y 256.127,Z 180.58,A -85,B 0,C 180,E1 -18512.194,E2 -18512.194} C_VEL
LIN {X 0,Y 256.131,Z 180.58,A -85,B 0,C 180,E1 -18515.695,E2 -18515.695} C_VEL
LIN {X 0,Y 256.15,Z 180.576,A -85,B 0,C 180,E1 -18519.103,E2 -18519.103} C_VEL
LIN {X 0,Y 256.287,Z 180.559,A -85,B 0,C 180,E1 -18524.084,E2 -18524.084} C_VEL
LIN {X 0,Y 256.297,Z 180.559,A -85,B 0,C 180,E1 -18528.933,E2 -18528.933} C_VEL
LIN {X 0,Y 256.525,Z 180.527,A -85,B 0,C 180,E1 -18532.126,E2 -18532.126} C_VEL
LIN {X 0,Y 256.705,Z 180.506,A -85,B 0,C 180,E1 -18538.431,E2 -18538.431} C_VEL
LIN {X 0,Y 256.699,Z 180.507,A -85,B 0,C 180,E1 -18541.569,E2 -18541.569} C_VEL
LIN {X 0,Y 256.526,Z 180.527,A -85,B 0,C 180,E1 -18547.873,E2 -18547.873} C_VEL
LIN {X 0,Y 256.297,Z 180.559,A -85,B 0,C 180,E1 -18551.066,E2 -18551.066} C_VEL
LIN {X 0,Y 256.287,Z 180.559,A -85,B 0,C 180,E1 -18555.916,E2 -18555.916} C_VEL
LIN {X 0,Y 256.152,Z 180.576,A -85,B 0,C 180,E1 -18560.896,E2 -18560.896} C_VEL
LIN {X 0,Y 256.122,Z 180.577,A -85,B 0,C 180,E1 -18565.114,E2 -18565.114} C_VEL
LIN {X 0,Y 256.044,Z 180.59,A -85,B 0,C 180,E1 -18569.608,E2 -18569.608} C_VEL
LIN {X 0,Y 256.072,Z 180.585,A -85,B 0,C 180,E1 -18573.292,E2 -18573.292} C_VEL
LIN {X 0,Y 256.118,Z 180.58,A -85,B 0,C 180,E1 -18577.277,E2 -18577.277} C_VEL
LIN {X 0,Y 256.065,Z 180.587,A -85,B 0,C 180,E1 -18581.201,E2 -18581.201} C_VEL
LIN {X 0,Y 256.055,Z 180.592,A -85,B 0,C 180,E1 -18585.531,E2 -18585.531} C_VEL
LIN {X 0,Y 256.047,Z 180.589,A -85,B 0,C 180,E1 -18588.799,E2 -18588.799} C_VEL
LIN {X 0,Y 256.123,Z 180.579,A -85,B 0,C 180,E1 -18592.87,E2 -18592.87} C_VEL
LIN {X 0,Y 256.061,Z 180.588,A -85,B 0,C 180,E1 -18596.71,E2 -18596.71} C_VEL
LIN {X 0,Y 256.108,Z 180.579,A -85,B 0,C 180,E1 -18600.403,E2 -18600.403} C_VEL
LIN {X 0,Y 256.184,Z 180.575,A -85,B 0,C 180,E1 -18604.864,E2 -18604.864} C_VEL
LIN {X 0,Y 256.164,Z 180.574,A -85,B 0,C 180,E1 -18609.108,E2 -18609.108} C_VEL
LIN {X 0,Y 256.298,Z 180.559,A -85,B 0,C 180,E1 -18614.088,E2 -18614.088} C_VEL
LIN {X 0,Y 256.309,Z 180.556,A -85,B 0,C 180,E1 -18618.937,E2 -18618.937} C_VEL
LIN {X 0,Y 256.54,Z 180.53,A -85,B 0,C 180,E1 -18622.13,E2 -18622.13} C_VEL
LIN {X 0,Y 256.71,Z 180.508,A -85,B 0,C 180,E1 -18628.434,E2 -18628.434} C_VEL
LIN {X 0,Y 256.709,Z 180.508,A -85,B 0,C 180,E1 -18631.571,E2 -18631.571} C_VEL
LIN {X 0,Y 256.543,Z 180.53,A -85,B 0,C 180,E1 -18637.875,E2 -18637.875} C_VEL
LIN {X 0,Y 256.313,Z 180.556,A -85,B 0,C 180,E1 -18641.068,E2 -18641.068} C_VEL
LIN {X 0,Y 256.304,Z 180.558,A -85,B 0,C 180,E1 -18645.917,E2 -18645.917} C_VEL
LIN {X 0,Y 256.153,Z 180.575,A -85,B 0,C 180,E1 -18650.899,E2 -18650.899} C_VEL
LIN {X 0,Y 256.089,Z 180.587,A -85,B 0,C 180,E1 -18655.091,E2 -18655.091} C_VEL
LIN {X 0,Y 256.094,Z 180.583,A -85,B 0,C 180,E1 -18658.577,E2 -18658.577} C_VEL
LIN {X 0,Y 256.079,Z 180.584,A -85,B 0,C 180,E1 -18661.703,E2 -18661.703} C_VEL
LIN {X 0,Y 256.086,Z 180.585,A -85,B 0,C 180,E1 -18665.195,E2 -18665.195} C_VEL
LIN {X 0,Y 256.117,Z 180.579,A -85,B 0,C 180,E1 -18667.271,E2 -18667.271} C_VEL
LIN {X 0,Y 256.024,Z 180.592,A -85,B 0,C 180,E1 -18671.212,E2 -18671.212} C_VEL
LIN {X 0,Y 256.059,Z 180.586,A -85,B 0,C 180,E1 -18675.533,E2 -18675.533} C_VEL
LIN {X 0,Y 256.065,Z 180.587,A -85,B 0,C 180,E1 -18678.799,E2 -18678.799} C_VEL
LIN {X 0,Y 256.213,Z 180.569,A -85,B 0,C 180,E1 -18683.861,E2 -18683.861} C_VEL
LIN {X 0,Y 256.285,Z 180.636,A -85,B 0,C 180,E1 -18684.719,E2 -18684.719} C_VEL
LIN {X 0,Y 257.166,Z 185.411,A -85,B 0,C 180,E1 -18687.91,E2 -18687.91} C_VEL
LIN {X 0,Y 257.051,Z 189.464,A -85,B 0,C 180,E1 -18690.519,E2 -18690.519} C_VEL
LIN {X 0,Y 256.153,Z 196.409,A -85,B 0,C 180,E1 -18694.883,E2 -18694.883} C_VEL
LIN {X 0,Y 255.484,Z 203.498,A -85,B 0,C 180,E1 -18699.28,E2 -18699.28} C_VEL
LIN {X 0,Y 254.93,Z 209.854,A -85,B 0,C 180,E1 -18703.174,E2 -18703.174} C_VEL
LIN {X 0,Y 254.671,Z 216.893,A -85,B 0,C 180,E1 -18707.448,E2 -18707.448} C_VEL
LIN {X 0,Y 255.247,Z 228.358,A -85,B 0,C 180,E1 -18708.485,E2 -18708.485} C_VEL
LIN {X 0,Y 255.954,Z 237.428,A -85,B 0,C 180,E1 -18709.519,E2 -18709.519} C_VEL
LIN {X 0,Y 255.512,Z 248.31,A -85,B 0,C 180,E1 -18711.1,E2 -18711.1} C_VEL
LIN {X 0,Y 255.029,Z 257.534,A -85,B 0,C 180,E1 -18712.795,E2 -18712.795} C_VEL
LIN {X 0,Y 254.737,Z 266.412,A -85,B 0,C 180,E1 -18714.856,E2 -18714.856} C_VEL
LIN {X 0,Y 254.375,Z 273.129,A -85,B 0,C 180,E1 -18716.833,E2 -18716.833} C_VEL
LIN {X 0,Y 254.211,Z 277.477,A -85,B 0,C 180,E1 -18718.416,E2 -18718.416} C_VEL
LIN {X 0,Y 254.258,Z 282.604,A -85,B 0,C 180,E1 -18720.792,E2 -18720.792} C_VEL
LIN {X 0,Y 254.69,Z 286.22,A -85,B 0,C 180,E1 -18723.164,E2 -18723.164} C_VEL
LIN {X 0,Y 255.227,Z 287.874,A -85,B 0,C 180,E1 -18724.739,E2 -18724.739} C_VEL
LIN {X 0,Y 255.989,Z 288.916,A -85,B 0,C 180,E1 -18726.305,E2 -18726.305} C_VEL
LIN {X 0,Y 256.649,Z 289.41,A -85,B 0,C 180,E1 -18727.87,E2 -18727.87} C_VEL
LIN {X 0,Y 257.67,Z 289.354,A -85,B 0,C 180,E1 -18729.419,E2 -18729.419} C_VEL
LIN {X 0,Y 258.88,Z 288.72,A -85,B 0,C 180,E1 -18730.955,E2 -18730.955} C_VEL
LIN {X 0,Y 260.435,Z 287.522,A -85,B 0,C 180,E1 -18732.468,E2 -18732.468} C_VEL
LIN {X 0,Y 263.035,Z 284.707,A -85,B 0,C 180,E1 -18734.704,E2 -18734.704} C_VEL
LIN {X 0,Y 266.191,Z 280.508,A -85,B 0,C 180,E1 -18736.883,E2 -18736.883} C_VEL
LIN {X 0,Y 269.759,Z 274.862,A -85,B 0,C 180,E1 -18739.006,E2 -18739.006} C_VEL
LIN {X 0,Y 272.803,Z 269.046,A -85,B 0,C 180,E1 -18740.746,E2 -18740.746} C_VEL
LIN {X 0,Y 274.204,Z 261.832,A -85,B 0,C 180,E1 -18743.009,E2 -18743.009} C_VEL
LIN {X 0,Y 274.616,Z 254.578,A -85,B 0,C 180,E1 -18745.249,E2 -18745.249} C_VEL
LIN {X 0,Y 274.161,Z 245.75,A -85,B 0,C 180,E1 -18748.094,E2 -18748.094} C_VEL
LIN {X 0,Y 274.014,Z 244.329,A -85,B 0,C 180,E1 -18748.569,E2 -18748.569} C_VEL
LIN {X 0,Y 273.205,Z 241.857,A -85,B 0,C 180,E1 -18749.68,E2 -18749.68} C_VEL
LIN {X 0,Y 271.926,Z 240.145,A -85,B 0,C 180,E1 -18750.846,E2 -18750.846} C_VEL
LIN {X 0,Y 268.235,Z 237.084,A -85,B 0,C 180,E1 -18754.098,E2 -18754.098} C_VEL
LIN {X 0,Y 267.653,Z 236.162,A -85,B 0,C 180,E1 -18754.926,E2 -18754.926} C_VEL
LIN {X 0,Y 266.637,Z 232.842,A -85,B 0,C 180,E1 -18757.742,E2 -18757.742} C_VEL
LIN {X 0,Y 266.025,Z 231.572,A -85,B 0,C 180,E1 -18759.989,E2 -18759.989} C_VEL
LIN {X 0,Y 265.961,Z 231.209,A -85,B 0,C 180,E1 -18763.397,E2 -18763.397} C_VEL
LIN {X 0,Y 267.141,Z 232.458,A -85,B 0,C 180,E1 -18766.839,E2 -18766.839} C_VEL
LIN {X 0,Y 267.921,Z 233.793,A -85,B 0,C 180,E1 -18768.319,E2 -18768.319} C_VEL
LIN {X 0,Y 270.531,Z 238.613,A -85,B 0,C 180,E1 -18771.853,E2 -18771.853} C_VEL
LIN {X 0,Y 272.644,Z 243.441,A -85,B 0,C 180,E1 -18774.233,E2 -18774.233} C_VEL
LIN {X 0,Y 273.907,Z 246.914,A -85,B 0,C 180,E1 -18775.631,E2 -18775.631} C_VEL
LIN {X 0,Y 274.212,Z 248.542,A -85,B 0,C 180,E1 -18776.149,E2 -18776.149} C_VEL
LIN {X 0,Y 273.906,Z 257.329,A -85,B 0,C 180,E1 -18778.244,E2 -18778.244} C_VEL
LIN {X 0,Y 272.674,Z 266.343,A -85,B 0,C 180,E1 -18780.294,E2 -18780.294} C_VEL
LIN {X 0,Y 271.891,Z 269.613,A -85,B 0,C 180,E1 -18781.007,E2 -18781.007} C_VEL
LIN {X 0,Y 267.266,Z 279.653,A -85,B 0,C 180,E1 -18783.023,E2 -18783.023} C_VEL
LIN {X 0,Y 262.892,Z 287.92,A -85,B 0,C 180,E1 -18785.097,E2 -18785.097} C_VEL
LIN {X 0,Y 259.021,Z 294.693,A -85,B 0,C 180,E1 -18787.252,E2 -18787.252} C_VEL
LIN {X 0,Y 256.202,Z 299.359,A -85,B 0,C 180,E1 -18789.106,E2 -18789.106} C_VEL
LIN {X 0,Y 253.576,Z 303.928,A -85,B 0,C 180,E1 -18791.412,E2 -18791.412} C_VEL
LIN {X 0,Y 251.206,Z 307.533,A -85,B 0,C 180,E1 -18793.751,E2 -18793.751} C_VEL
LIN {X 0,Y 249.881,Z 309.429,A -85,B 0,C 180,E1 -18795.335,E2 -18795.335} C_VEL
LIN {X 0,Y 248.144,Z 311.996,A -85,B 0,C 180,E1 -18798.563,E2 -18798.563} C_VEL
LIN {X 0,Y 247.608,Z 312.736,A -85,B 0,C 180,E1 -18800.192,E2 -18800.192} C_VEL
LIN {X 0,Y 247.116,Z 313.021,A -85,B 0,C 180,E1 -18803.465,E2 -18803.465} C_VEL
LIN {X 0,Y 247.193,Z 312.607,A -85,B 0,C 180,E1 -18805.105,E2 -18805.105} C_VEL
LIN {X 0,Y 247.182,Z 311.773,A -85,B 0,C 180,E1 -18806.738,E2 -18806.738} C_VEL
LIN {X 0,Y 247.571,Z 310.534,A -85,B 0,C 180,E1 -18808.371,E2 -18808.371} C_VEL
LIN {X 0,Y 247.804,Z 307.785,A -85,B 0,C 180,E1 -18810.81,E2 -18810.81} C_VEL
LIN {X 0,Y 247.79,Z 303.855,A -85,B 0,C 180,E1 -18813.249,E2 -18813.249} C_VEL
LIN {X 0,Y 247.86,Z 298.63,A -85,B 0,C 180,E1 -18815.693,E2 -18815.693} C_VEL
LIN {X 0,Y 247.981,Z 291.817,A -85,B 0,C 180,E1 -18818.144,E2 -18818.144} C_VEL
LIN {X 0,Y 248.282,Z 283.179,A -85,B 0,C 180,E1 -18820.6,E2 -18820.6} C_VEL
LIN {X 0,Y 248.79,Z 274.127,A -85,B 0,C 180,E1 -18822.643,E2 -18822.643} C_VEL
LIN {X 0,Y 249.37,Z 265.276,A -85,B 0,C 180,E1 -18824.274,E2 -18824.274} C_VEL
LIN {X 0,Y 250.165,Z 254.335,A -85,B 0,C 180,E1 -18825.894,E2 -18825.894} C_VEL
LIN {X 0,Y 250.409,Z 246.328,A -85,B 0,C 180,E1 -18826.856,E2 -18826.856} C_VEL
LIN {X 0,Y 249.262,Z 233.382,A -85,B 0,C 180,E1 -18828.065,E2 -18828.065} C_VEL
LIN {X 0,Y 248.743,Z 219.966,A -85,B 0,C 180,E1 -18828.958,E2 -18828.958} C_VEL
LIN {X 0,Y 250.59,Z 207.948,A -85,B 0,C 180,E1 -18834.875,E2 -18834.875} C_VEL
LIN {X 0,Y 252.048,Z 201.001,A -85,B 0,C 180,E1 -18838.292,E2 -18838.292} C_VEL
LIN {X 0,Y 252.344,Z 199.239,A -85,B 0,C 180,E1 -18839.166,E2 -18839.166} C_VEL
LIN {X 0,Y 251.806,Z 195.52,A -85,B 0,C 180,E1 -18841.083,E2 -18841.083} C_VEL
LIN {X 0,Y 249.949,Z 185.95,A -85,B 0,C 180,E1 -18846.187,E2 -18846.187} C_VEL
LIN {X 0,Y 249.118,Z 181.453,A -85,B 0,C 180,E1 -18848.748,E2 -18848.748} C_VEL
LIN {X 0,Y 249.011,Z 181.468,A -85,B 0,C 180,E1 -18852.792,E2 -18852.792} C_VEL
LIN {X 0,Y 249.054,Z 181.457,A -85,B 0,C 180,E1 -18857.37,E2 -18857.37} C_VEL
LIN {X 0,Y 249.043,Z 181.461,A -85,B 0,C 180,E1 -18861.622,E2 -18861.622} C_VEL
LIN {X 0,Y 249.052,Z 181.459,A -85,B 0,C 180,E1 -18865.64,E2 -18865.64} C_VEL
LIN {X 0,Y 249.037,Z 181.463,A -85,B 0,C 180,E1 -18869.471,E2 -18869.471} C_VEL
LIN {X 0,Y 249.057,Z 181.458,A -85,B 0,C 180,E1 -18873.16,E2 -18873.16} C_VEL
LIN {X 0,Y 249.049,Z 181.46,A -85,B 0,C 180,E1 -18876.729,E2 -18876.729} C_VEL
LIN {X 0,Y 249.096,Z 181.455,A -85,B 0,C 180,E1 -18880.21,E2 -18880.21} C_VEL
LIN {X 0,Y 249.23,Z 181.44,A -85,B 0,C 180,E1 -18883.621,E2 -18883.621} C_VEL
LIN {X 0,Y 249.24,Z 181.436,A -85,B 0,C 180,E1 -18888.616,E2 -18888.616} C_VEL
LIN {X 0,Y 249.467,Z 181.407,A -85,B 0,C 180,E1 -18891.902,E2 -18891.902} C_VEL
LIN {X 0,Y 249.429,Z 181.415,A -85,B 0,C 180,E1 -18896.769,E2 -18896.769} C_VEL
LIN {X 0,Y 249.714,Z 181.375,A -85,B 0,C 180,E1 -18900,E2 -18900} C_VEL
LIN {X 0,Y 249.419,Z 181.416,A -85,B 0,C 180,E1 -18903.23,E2 -18903.23} C_VEL
LIN {X 0,Y 249.468,Z 181.407,A -85,B 0,C 180,E1 -18908.097,E2 -18908.097} C_VEL
LIN {X 0,Y 249.24,Z 181.436,A -85,B 0,C 180,E1 -18911.384,E2 -18911.384} C_VEL
LIN {X 0,Y 249.229,Z 181.44,A -85,B 0,C 180,E1 -18916.379,E2 -18916.379} C_VEL
LIN {X 0,Y 249.072,Z 181.458,A -85,B 0,C 180,E1 -18921.519,E2 -18921.519} C_VEL
LIN {X 0,Y 249.074,Z 181.455,A -85,B 0,C 180,E1 -18925.462,E2 -18925.462} C_VEL
LIN {X 0,Y 249.027,Z 181.463,A -85,B 0,C 180,E1 -18928.976,E2 -18928.976} C_VEL
LIN {X 0,Y 249.021,Z 181.464,A -85,B 0,C 180,E1 -18932.427,E2 -18932.427} C_VEL
LIN {X 0,Y 249.059,Z 181.459,A -85,B 0,C 180,E1 -18936.341,E2 -18936.341} C_VEL
LIN {X 0,Y 249.022,Z 181.463,A -85,B 0,C 180,E1 -18940.475,E2 -18940.475} C_VEL
LIN {X 0,Y 249.001,Z 181.466,A -85,B 0,C 180,E1 -18944.88,E2 -18944.88} C_VEL
LIN {X 0,Y 249.01,Z 181.469,A -85,B 0,C 180,E1 -18947.366,E2 -18947.366} C_VEL
LIN {X 0,Y 249.036,Z 181.46,A -85,B 0,C 180,E1 -18952.203,E2 -18952.203} C_VEL
LIN {X 0,Y 249.037,Z 181.463,A -85,B 0,C 180,E1 -18955.642,E2 -18955.642} C_VEL
LIN {X 0,Y 249.046,Z 181.459,A -85,B 0,C 180,E1 -18959.476,E2 -18959.476} C_VEL
LIN {X 0,Y 249.069,Z 181.46,A -85,B 0,C 180,E1 -18963.165,E2 -18963.165} C_VEL
LIN {X 0,Y 249.076,Z 181.46,A -85,B 0,C 180,E1 -18966.735,E2 -18966.735} C_VEL
LIN {X 0,Y 249.108,Z 181.453,A -85,B 0,C 180,E1 -18970.214,E2 -18970.214} C_VEL
LIN {X 0,Y 249.24,Z 181.436,A -85,B 0,C 180,E1 -18973.625,E2 -18973.625} C_VEL
LIN {X 0,Y 249.252,Z 181.437,A -85,B 0,C 180,E1 -18978.619,E2 -18978.619} C_VEL
LIN {X 0,Y 249.484,Z 181.408,A -85,B 0,C 180,E1 -18981.906,E2 -18981.906} C_VEL
LIN {X 0,Y 249.437,Z 181.411,A -85,B 0,C 180,E1 -18986.772,E2 -18986.772} C_VEL
LIN {X 0,Y 249.672,Z 181.384,A -85,B 0,C 180,E1 -18988.39,E2 -18988.39} C_VEL
LIN {X 0,Y 249.671,Z 181.385,A -85,B 0,C 180,E1 -18991.616,E2 -18991.616} C_VEL
LIN {X 0,Y 249.463,Z 181.409,A -85,B 0,C 180,E1 -18996.473,E2 -18996.473} C_VEL
LIN {X 0,Y 249.428,Z 181.416,A -85,B 0,C 180,E1 -18999.736,E2 -18999.736} C_VEL
LIN {X 0,Y 249.209,Z 181.439,A -85,B 0,C 180,E1 -19004.706,E2 -19004.706} C_VEL
LIN {X 0,Y 249.141,Z 181.449,A -85,B 0,C 180,E1 -19008.08,E2 -19008.08} C_VEL
LIN {X 0,Y 249.083,Z 181.457,A -85,B 0,C 180,E1 -19011.521,E2 -19011.521} C_VEL
LIN {X 0,Y 249.051,Z 181.462,A -85,B 0,C 180,E1 -19015.443,E2 -19015.443} C_VEL
LIN {X 0,Y 249.041,Z 181.463,A -85,B 0,C 180,E1 -19018.975,E2 -19018.975} C_VEL
LIN {X 0,Y 249.032,Z 181.463,A -85,B 0,C 180,E1 -19022.428,E2 -19022.428} C_VEL
LIN {X 0,Y 249.051,Z 181.461,A -85,B 0,C 180,E1 -19026.344,E2 -19026.344} C_VEL
LIN {X 0,Y 248.984,Z 181.47,A -85,B 0,C 180,E1 -19030.485,E2 -19030.485} C_VEL
LIN {X 0,Y 248.996,Z 181.467,A -85,B 0,C 180,E1 -19034.884,E2 -19034.884} C_VEL
LIN {X 0,Y 249.025,Z 181.461,A -85,B 0,C 180,E1 -19037.365,E2 -19037.365} C_VEL
LIN {X 0,Y 249.041,Z 181.462,A -85,B 0,C 180,E1 -19041.622,E2 -19041.622} C_VEL
LIN {X 0,Y 249.232,Z 181.477,A -85,B 0,C 180,E1 -19044.652,E2 -19044.652} C_VEL
LIN {X 0,Y 250.079,Z 185.943,A -85,B 0,C 180,E1 -19047.727,E2 -19047.727} C_VEL
LIN {X 0,Y 250.128,Z 188.798,A -85,B 0,C 180,E1 -19049.618,E2 -19049.618} C_VEL
LIN {X 0,Y 249.262,Z 195.505,A -85,B 0,C 180,E1 -19053.943,E2 -19053.943} C_VEL
LIN {X 0,Y 248.515,Z 202.556,A -85,B 0,C 180,E1 -19058.43,E2 -19058.43} C_VEL
LIN {X 0,Y 247.897,Z 209.296,A -85,B 0,C 180,E1 -19062.682,E2 -19062.682} C_VEL
LIN {X 0,Y 247.579,Z 216.936,A -85,B 0,C 180,E1 -19067.447,E2 -19067.447} C_VEL
LIN {X 0,Y 248.168,Z 228.759,A -85,B 0,C 180,E1 -19068.566,E2 -19068.566} C_VEL
LIN {X 0,Y 248.875,Z 237.759,A -85,B 0,C 180,E1 -19069.629,E2 -19069.629} C_VEL
LIN {X 0,Y 248.414,Z 248.556,A -85,B 0,C 180,E1 -19071.253,E2 -19071.253} C_VEL
LIN {X 0,Y 247.906,Z 258.025,A -85,B 0,C 180,E1 -19073.054,E2 -19073.054} C_VEL
LIN {X 0,Y 247.645,Z 266.631,A -85,B 0,C 180,E1 -19075.116,E2 -19075.116} C_VEL
LIN {X 0,Y 247.261,Z 273.348,A -85,B 0,C 180,E1 -19077.149,E2 -19077.149} C_VEL
LIN {X 0,Y 247.107,Z 278.711,A -85,B 0,C 180,E1 -19079.185,E2 -19079.185} C_VEL
LIN {X 0,Y 247.288,Z 283.613,A -85,B 0,C 180,E1 -19081.629,E2 -19081.629} C_VEL
LIN {X 0,Y 247.622,Z 286.042,A -85,B 0,C 180,E1 -19083.254,E2 -19083.254} C_VEL
LIN {X 0,Y 248.17,Z 287.88,A -85,B 0,C 180,E1 -19084.874,E2 -19084.874} C_VEL
LIN {X 0,Y 248.945,Z 289.145,A -85,B 0,C 180,E1 -19086.484,E2 -19086.484} C_VEL
LIN {X 0,Y 249.641,Z 289.842,A -85,B 0,C 180,E1 -19088.092,E2 -19088.092} C_VEL
LIN {X 0,Y 250.696,Z 289.97,A -85,B 0,C 180,E1 -19089.684,E2 -19089.684} C_VEL
LIN {X 0,Y 251.973,Z 289.573,A -85,B 0,C 180,E1 -19091.259,E2 -19091.259} C_VEL
LIN {X 0,Y 253.596,Z 288.602,A -85,B 0,C 180,E1 -19092.809,E2 -19092.809} C_VEL
LIN {X 0,Y 256.288,Z 286.126,A -85,B 0,C 180,E1 -19095.101,E2 -19095.101} C_VEL
LIN {X 0,Y 259.587,Z 282.354,A -85,B 0,C 180,E1 -19097.326,E2 -19097.326} C_VEL
LIN {X 0,Y 263.287,Z 277.192,A -85,B 0,C 180,E1 -19099.492,E2 -19099.492} C_VEL
LIN {X 0,Y 266.617,Z 271.762,A -85,B 0,C 180,E1 -19101.251,E2 -19101.251} C_VEL
LIN {X 0,Y 268.205,Z 266.188,A -85,B 0,C 180,E1 -19103.145,E2 -19103.145} C_VEL
LIN {X 0,Y 269.062,Z 259.948,A -85,B 0,C 180,E1 -19105.255,E2 -19105.255} C_VEL
LIN {X 0,Y 269.348,Z 251.911,A -85,B 0,C 180,E1 -19108.013,E2 -19108.013} C_VEL
LIN {X 0,Y 269.006,Z 244.49,A -85,B 0,C 180,E1 -19110.784,E2 -19110.784} C_VEL
LIN {X 0,Y 268.625,Z 240.931,A -85,B 0,C 180,E1 -19112.305,E2 -19112.305} C_VEL
LIN {X 0,Y 267.989,Z 236.895,A -85,B 0,C 180,E1 -19114.339,E2 -19114.339} C_VEL
LIN {X 0,Y 267.653,Z 236.162,A -85,B 0,C 180,E1 -19114.926,E2 -19114.926} C_VEL
LIN {X 0,Y 266.742,Z 235.311,A -85,B 0,C 180,E1 -19116.165,E2 -19116.165} C_VEL
LIN {X 0,Y 265.545,Z 235.473,A -85,B 0,C 180,E1 -19117.421,E2 -19117.421} C_VEL
LIN {X 0,Y 262.846,Z 237.442,A -85,B 0,C 180,E1 -19120.834,E2 -19120.834} C_VEL
LIN {X 0,Y 262.678,Z 237.554,A -85,B 0,C 180,E1 -19121.71,E2 -19121.71} C_VEL
LIN {X 0,Y 262.934,Z 237.711,A -85,B 0,C 180,E1 -19124.024,E2 -19124.024} C_VEL
LIN {X 0,Y 263.645,Z 238.451,A -85,B 0,C 180,E1 -19126.123,E2 -19126.123} C_VEL
LIN {X 0,Y 264.69,Z 240.335,A -85,B 0,C 180,E1 -19128.407,E2 -19128.407} C_VEL
LIN {X 0,Y 266.5,Z 244.008,A -85,B 0,C 180,E1 -19131.255,E2 -19131.255} C_VEL
LIN {X 0,Y 268.632,Z 249.633,A -85,B 0,C 180,E1 -19134.197,E2 -19134.197} C_VEL
LIN {X 0,Y 269.472,Z 252.782,A -85,B 0,C 180,E1 -19135.47,E2 -19135.47} C_VEL
LIN {X 0,Y 268.614,Z 261.547,A -85,B 0,C 180,E1 -19137.717,E2 -19137.717} C_VEL
LIN {X 0,Y 267.123,Z 269.128,A -85,B 0,C 180,E1 -19139.569,E2 -19139.569} C_VEL
LIN {X 0,Y 266.056,Z 272.382,A -85,B 0,C 180,E1 -19140.309,E2 -19140.309} C_VEL
LIN {X 0,Y 261.139,Z 281.778,A -85,B 0,C 180,E1 -19142.336,E2 -19142.336} C_VEL
LIN {X 0,Y 256.602,Z 289.536,A -85,B 0,C 180,E1 -19144.443,E2 -19144.443} C_VEL
LIN {X 0,Y 251.955,Z 296.795,A -85,B 0,C 180,E1 -19147.011,E2 -19147.011} C_VEL
LIN {X 0,Y 248.653,Z 301.766,A -85,B 0,C 180,E1 -19149.308,E2 -19149.308} C_VEL
LIN {X 0,Y 245.211,Z 306.785,A -85,B 0,C 180,E1 -19152.483,E2 -19152.483} C_VEL
LIN {X 0,Y 243.026,Z 309.495,A -85,B 0,C 180,E1 -19154.911,E2 -19154.911} C_VEL
LIN {X 0,Y 241.923,Z 310.831,A -85,B 0,C 180,E1 -19156.559,E2 -19156.559} C_VEL
LIN {X 0,Y 240.601,Z 312.337,A -85,B 0,C 180,E1 -19159.904,E2 -19159.904} C_VEL
LIN {X 0,Y 240.052,Z 312.373,A -85,B 0,C 180,E1 -19163.272,E2 -19163.272} C_VEL
LIN {X 0,Y 240.138,Z 311.801,A -85,B 0,C 180,E1 -19164.96,E2 -19164.96} C_VEL
LIN {X 0,Y 240.543,Z 309.478,A -85,B 0,C 180,E1 -19168.323,E2 -19168.323} C_VEL
LIN {X 0,Y 240.823,Z 306.528,A -85,B 0,C 180,E1 -19170.833,E2 -19170.833} C_VEL
LIN {X 0,Y 240.796,Z 302.328,A -85,B 0,C 180,E1 -19173.344,E2 -19173.344} C_VEL
LIN {X 0,Y 240.879,Z 296.789,A -85,B 0,C 180,E1 -19175.858,E2 -19175.858} C_VEL
LIN {X 0,Y 240.98,Z 291.134,A -85,B 0,C 180,E1 -19177.908,E2 -19177.908} C_VEL
LIN {X 0,Y 241.147,Z 283.843,A -85,B 0,C 180,E1 -19180.068,E2 -19180.068} C_VEL
LIN {X 0,Y 241.637,Z 275.082,A -85,B 0,C 180,E1 -19182.17,E2 -19182.17} C_VEL
LIN {X 0,Y 242.28,Z 265.36,A -85,B 0,C 180,E1 -19184.057,E2 -19184.057} C_VEL
LIN {X 0,Y 243.035,Z 254.598,A -85,B 0,C 180,E1 -19185.727,E2 -19185.727} C_VEL
LIN {X 0,Y 243.411,Z 248.064,A -85,B 0,C 180,E1 -19186.563,E2 -19186.563} C_VEL
LIN {X 0,Y 242.403,Z 236.219,A -85,B 0,C 180,E1 -19187.772,E2 -19187.772} C_VEL
LIN {X 0,Y 241.656,Z 223.848,A -85,B 0,C 180,E1 -19188.709,E2 -19188.709} C_VEL
LIN {X 0,Y 241.658,Z 219.889,A -85,B 0,C 180,E1 -19188.984,E2 -19188.984} C_VEL
LIN {X 0,Y 243.415,Z 208.586,A -85,B 0,C 180,E1 -19194.746,E2 -19194.746} C_VEL
LIN {X 0,Y 245.224,Z 199.928,A -85,B 0,C 180,E1 -19199.154,E2 -19199.154} C_VEL
LIN {X 0,Y 244.724,Z 196.229,A -85,B 0,C 180,E1 -19201.123,E2 -19201.123} C_VEL
LIN {X 0,Y 243.021,Z 187.458,A -85,B 0,C 180,E1 -19205.929,E2 -19205.929} C_VEL
LIN {X 0,Y 242.05,Z 182.332,A -85,B 0,C 180,E1 -19208.903,E2 -19208.903} C_VEL
LIN {X 0,Y 241.936,Z 182.346,A -85,B 0,C 180,E1 -19213.429,E2 -19213.429} C_VEL
LIN {X 0,Y 241.983,Z 182.341,A -85,B 0,C 180,E1 -19216.555,E2 -19216.555} C_VEL
LIN {X 0,Y 241.999,Z 182.342,A -85,B 0,C 180,E1 -19220.289,E2 -19220.289} C_VEL
LIN {X 0,Y 242.027,Z 182.335,A -85,B 0,C 180,E1 -19224.496,E2 -19224.496} C_VEL
LIN {X 0,Y 241.964,Z 182.344,A -85,B 0,C 180,E1 -19228.478,E2 -19228.478} C_VEL
LIN {X 0,Y 241.99,Z 182.34,A -85,B 0,C 180,E1 -19232.31,E2 -19232.31} C_VEL
LIN {X 0,Y 242.029,Z 182.337,A -85,B 0,C 180,E1 -19236.013,E2 -19236.013} C_VEL
LIN {X 0,Y 242.024,Z 182.339,A -85,B 0,C 180,E1 -19239.607,E2 -19239.607} C_VEL
LIN {X 0,Y 242.151,Z 182.319,A -85,B 0,C 180,E1 -19243.277,E2 -19243.277} C_VEL
LIN {X 0,Y 242.174,Z 182.317,A -85,B 0,C 180,E1 -19248.279,E2 -19248.279} C_VEL
LIN {X 0,Y 242.414,Z 182.287,A -85,B 0,C 180,E1 -19251.665,E2 -19251.665} C_VEL
LIN {X 0,Y 242.25,Z 182.31,A -85,B 0,C 180,E1 -19255.007,E2 -19255.007} C_VEL
LIN {X 0,Y 242.627,Z 182.26,A -85,B 0,C 180,E1 -19258.34,E2 -19258.34} C_VEL
LIN {X 0,Y 242.622,Z 182.26,A -85,B 0,C 180,E1 -19261.66,E2 -19261.66} C_VEL
LIN {X 0,Y 242.413,Z 182.289,A -85,B 0,C 180,E1 -19266.77,E2 -19266.77} C_VEL
LIN {X 0,Y 242.301,Z 182.3,A -85,B 0,C 180,E1 -19270.022,E2 -19270.022} C_VEL
LIN {X 0,Y 242.154,Z 182.319,A -85,B 0,C 180,E1 -19275.141,E2 -19275.141} C_VEL
LIN {X 0,Y 242.061,Z 182.333,A -85,B 0,C 180,E1 -19278.625,E2 -19278.625} C_VEL
LIN {X 0,Y 241.994,Z 182.343,A -85,B 0,C 180,E1 -19282.182,E2 -19282.182} C_VEL
LIN {X 0,Y 242.02,Z 182.336,A -85,B 0,C 180,E1 -19285.822,E2 -19285.822} C_VEL
LIN {X 0,Y 241.958,Z 182.345,A -85,B 0,C 180,E1 -19289.59,E2 -19289.59} C_VEL
LIN {X 0,Y 241.979,Z 182.341,A -85,B 0,C 180,E1 -19293.493,E2 -19293.493} C_VEL
LIN {X 0,Y 241.992,Z 182.342,A -85,B 0,C 180,E1 -19297.581,E2 -19297.581} C_VEL
LIN {X 0,Y 241.943,Z 182.345,A -85,B 0,C 180,E1 -19301.921,E2 -19301.921} C_VEL
LIN {X 0,Y 241.929,Z 182.347,A -85,B 0,C 180,E1 -19306.573,E2 -19306.573} C_VEL
LIN {X 0,Y 241.948,Z 182.343,A -85,B 0,C 180,E1 -19310.283,E2 -19310.283} C_VEL
LIN {X 0,Y 241.981,Z 182.341,A -85,B 0,C 180,E1 -19314.492,E2 -19314.492} C_VEL
LIN {X 0,Y 241.969,Z 182.342,A -85,B 0,C 180,E1 -19318.483,E2 -19318.483} C_VEL
LIN {X 0,Y 242.004,Z 182.338,A -85,B 0,C 180,E1 -19322.316,E2 -19322.316} C_VEL
LIN {X 0,Y 242.054,Z 182.332,A -85,B 0,C 180,E1 -19326.019,E2 -19326.019} C_VEL
LIN {X 0,Y 242.035,Z 182.332,A -85,B 0,C 180,E1 -19329.611,E2 -19329.611} C_VEL
LIN {X 0,Y 242.161,Z 182.319,A -85,B 0,C 180,E1 -19333.281,E2 -19333.281} C_VEL
LIN {X 0,Y 242.186,Z 182.316,A -85,B 0,C 180,E1 -19338.283,E2 -19338.283} C_VEL
LIN {X 0,Y 242.435,Z 182.285,A -85,B 0,C 180,E1 -19341.669,E2 -19341.669} C_VEL
LIN {X 0,Y 242.261,Z 182.304,A -85,B 0,C 180,E1 -19345.01,E2 -19345.01} C_VEL
LIN {X 0,Y 242.633,Z 182.262,A -85,B 0,C 180,E1 -19348.343,E2 -19348.343} C_VEL
LIN {X 0,Y 242.632,Z 182.262,A -85,B 0,C 180,E1 -19351.662,E2 -19351.662} C_VEL
LIN {X 0,Y 242.436,Z 182.284,A -85,B 0,C 180,E1 -19356.661,E2 -19356.661} C_VEL
LIN {X 0,Y 242.349,Z 182.296,A -85,B 0,C 180,E1 -19360.023,E2 -19360.023} C_VEL
LIN {X 0,Y 242.171,Z 182.318,A -85,B 0,C 180,E1 -19365.143,E2 -19365.143} C_VEL
LIN {X 0,Y 242.073,Z 182.329,A -85,B 0,C 180,E1 -19368.627,E2 -19368.627} C_VEL
LIN {X 0,Y 241.993,Z 182.337,A -85,B 0,C 180,E1 -19372.184,E2 -19372.184} C_VEL
LIN {X 0,Y 241.991,Z 182.34,A -85,B 0,C 180,E1 -19375.828,E2 -19375.828} C_VEL
LIN {X 0,Y 241.973,Z 182.339,A -85,B 0,C 180,E1 -19379.59,E2 -19379.59} C_VEL
LIN {X 0,Y 241.985,Z 182.341,A -85,B 0,C 180,E1 -19383.495,E2 -19383.495} C_VEL
LIN {X 0,Y 241.992,Z 182.337,A -85,B 0,C 180,E1 -19387.584,E2 -19387.584} C_VEL
LIN {X 0,Y 241.918,Z 182.349,A -85,B 0,C 180,E1 -19391.929,E2 -19391.929} C_VEL
LIN {X 0,Y 241.94,Z 182.346,A -85,B 0,C 180,E1 -19396.573,E2 -19396.573} C_VEL
LIN {X 0,Y 241.977,Z 182.345,A -85,B 0,C 180,E1 -19400.285,E2 -19400.285} C_VEL
LIN {X 0,Y 242.194,Z 182.398,A -85,B 0,C 180,E1 -19404.652,E2 -19404.652} C_VEL
LIN {X 0,Y 243.043,Z 186.977,A -85,B 0,C 180,E1 -19407.868,E2 -19407.868} C_VEL
LIN {X 0,Y 242.922,Z 190.461,A -85,B 0,C 180,E1 -19410.223,E2 -19410.223} C_VEL
LIN {X 0,Y 242.12,Z 196.457,A -85,B 0,C 180,E1 -19414.189,E2 -19414.189} C_VEL
LIN {X 0,Y 241.378,Z 203.384,A -85,B 0,C 180,E1 -19418.709,E2 -19418.709} C_VEL
LIN {X 0,Y 240.747,Z 210.063,A -85,B 0,C 180,E1 -19423.027,E2 -19423.027} C_VEL
LIN {X 0,Y 240.483,Z 217.042,A -85,B 0,C 180,E1 -19427.5,E2 -19427.5} C_VEL
LIN {X 0,Y 241.078,Z 228.958,A -85,B 0,C 180,E1 -19428.651,E2 -19428.651} C_VEL
LIN {X 0,Y 241.798,Z 237.955,A -85,B 0,C 180,E1 -19429.745,E2 -19429.745} C_VEL
LIN {X 0,Y 241.323,Z 248.708,A -85,B 0,C 180,E1 -19431.416,E2 -19431.416} C_VEL
LIN {X 0,Y 240.784,Z 258.264,A -85,B 0,C 180,E1 -19433.295,E2 -19433.295} C_VEL
LIN {X 0,Y 240.557,Z 266.783,A -85,B 0,C 180,E1 -19435.392,E2 -19435.392} C_VEL
LIN {X 0,Y 240.172,Z 273.51,A -85,B 0,C 180,E1 -19437.484,E2 -19437.484} C_VEL
LIN {X 0,Y 240.037,Z 277.92,A -85,B 0,C 180,E1 -19439.161,E2 -19439.161} C_VEL
LIN {X 0,Y 240.215,Z 283.135,A -85,B 0,C 180,E1 -19441.677,E2 -19441.677} C_VEL
LIN {X 0,Y 240.81,Z 286.885,A -85,B 0,C 180,E1 -19444.184,E2 -19444.184} C_VEL
LIN {X 0,Y 241.906,Z 289.271,A -85,B 0,C 180,E1 -19446.674,E2 -19446.674} C_VEL
LIN {X 0,Y 242.638,Z 290.183,A -85,B 0,C 180,E1 -19448.327,E2 -19448.327} C_VEL
LIN {X 0,Y 243.726,Z 290.54,A -85,B 0,C 180,E1 -19449.963,E2 -19449.963} C_VEL
LIN {X 0,Y 245.054,Z 290.338,A -85,B 0,C 180,E1 -19451.581,E2 -19451.581} C_VEL
LIN {X 0,Y 246.749,Z 289.607,A -85,B 0,C 180,E1 -19453.171,E2 -19453.171} C_VEL
LIN {X 0,Y 248.488,Z 288.355,A -85,B 0,C 180,E1 -19454.747,E2 -19454.747} C_VEL
LIN {X 0,Y 251.762,Z 285.399,A -85,B 0,C 180,E1 -19457.044,E2 -19457.044} C_VEL
LIN {X 0,Y 255.525,Z 281.157,A -85,B 0,C 180,E1 -19459.272,E2 -19459.272} C_VEL
LIN {X 0,Y 259.679,Z 275.502,A -85,B 0,C 180,E1 -19461.43,E2 -19461.43} C_VEL
LIN {X 0,Y 260.914,Z 273.379,A -85,B 0,C 180,E1 -19462.155,E2 -19462.155} C_VEL
LIN {X 0,Y 262.609,Z 268.049,A -85,B 0,C 180,E1 -19464.148,E2 -19464.148} C_VEL
LIN {X 0,Y 263.77,Z 261.632,A -85,B 0,C 180,E1 -19466.506,E2 -19466.506} C_VEL
LIN {X 0,Y 264.316,Z 254.841,A -85,B 0,C 180,E1 -19469.084,E2 -19469.084} C_VEL
LIN {X 0,Y 264.398,Z 248.476,A -85,B 0,C 180,E1 -19471.72,E2 -19471.72} C_VEL
LIN {X 0,Y 264.334,Z 245.931,A -85,B 0,C 180,E1 -19472.895,E2 -19472.895} C_VEL
LIN {X 0,Y 264.102,Z 243.125,A -85,B 0,C 180,E1 -19474.414,E2 -19474.414} C_VEL
LIN {X 0,Y 263.228,Z 239.038,A -85,B 0,C 180,E1 -19477.886,E2 -19477.886} C_VEL
LIN {X 0,Y 262.829,Z 237.93,A -85,B 0,C 180,E1 -19479.923,E2 -19479.923} C_VEL
LIN {X 0,Y 262.678,Z 237.554,A -85,B 0,C 180,E1 -19481.71,E2 -19481.71} C_VEL
LIN {X 0,Y 262.472,Z 238.112,A -85,B 0,C 180,E1 -19482.99,E2 -19482.99} C_VEL
LIN {X 0,Y 261.972,Z 239.673,A -85,B 0,C 180,E1 -19484.237,E2 -19484.237} C_VEL
LIN {X 0,Y 260.835,Z 245.435,A -85,B 0,C 180,E1 -19487.513,E2 -19487.513} C_VEL
LIN {X 0,Y 261.014,Z 246.559,A -85,B 0,C 180,E1 -19488.36,E2 -19488.36} C_VEL
LIN {X 0,Y 262.439,Z 249.676,A -85,B 0,C 180,E1 -19490.951,E2 -19490.951} C_VEL
LIN {X 0,Y 264.304,Z 255.62,A -85,B 0,C 180,E1 -19494.195,E2 -19494.195} C_VEL
LIN {X 0,Y 264.633,Z 257.114,A -85,B 0,C 180,E1 -19494.837,E2 -19494.837} C_VEL
LIN {X 0,Y 263.147,Z 265.877,A -85,B 0,C 180,E1 -19497.248,E2 -19497.248} C_VEL
LIN {X 0,Y 260.96,Z 273.501,A -85,B 0,C 180,E1 -19499.221,E2 -19499.221} C_VEL
LIN {X 0,Y 255.889,Z 282.519,A -85,B 0,C 180,E1 -19501.27,E2 -19501.27} C_VEL
LIN {X 0,Y 250.338,Z 291.073,A -85,B 0,C 180,E1 -19503.755,E2 -19503.755} C_VEL
LIN {X 0,Y 245.519,Z 297.856,A -85,B 0,C 180,E1 -19506.372,E2 -19506.372} C_VEL
LIN {X 0,Y 242.068,Z 302.466,A -85,B 0,C 180,E1 -19508.718,E2 -19508.718} C_VEL
LIN {X 0,Y 239.329,Z 306.084,A -85,B 0,C 180,E1 -19511.152,E2 -19511.152} C_VEL
LIN {X 0,Y 236.16,Z 309.55,A -85,B 0,C 180,E1 -19514.462,E2 -19514.462} C_VEL
LIN {X 0,Y 234.192,Z 311.479,A -85,B 0,C 180,E1 -19517.871,E2 -19517.871} C_VEL
LIN {X 0,Y 233.609,Z 311.916,A -85,B 0,C 180,E1 -19519.598,E2 -19519.598} C_VEL
LIN {X 0,Y 233.008,Z 311.614,A -85,B 0,C 180,E1 -19523.068,E2 -19523.068} C_VEL
LIN {X 0,Y 233.088,Z 310.93,A -85,B 0,C 180,E1 -19524.808,E2 -19524.808} C_VEL
LIN {X 0,Y 233.166,Z 309.825,A -85,B 0,C 180,E1 -19526.541,E2 -19526.541} C_VEL
LIN {X 0,Y 233.531,Z 308.303,A -85,B 0,C 180,E1 -19528.273,E2 -19528.273} C_VEL
LIN {X 0,Y 233.838,Z 305.126,A -85,B 0,C 180,E1 -19530.858,E2 -19530.858} C_VEL
LIN {X 0,Y 233.82,Z 300.678,A -85,B 0,C 180,E1 -19533.444,E2 -19533.444} C_VEL
LIN {X 0,Y 233.924,Z 294.875,A -85,B 0,C 180,E1 -19536.033,E2 -19536.033} C_VEL
LIN {X 0,Y 234.009,Z 288.912,A -85,B 0,C 180,E1 -19538.145,E2 -19538.145} C_VEL
LIN {X 0,Y 234.388,Z 279.555,A -85,B 0,C 180,E1 -19540.798,E2 -19540.798} C_VEL
LIN {X 0,Y 235.038,Z 268.81,A -85,B 0,C 180,E1 -19543.176,E2 -19543.176} C_VEL
LIN {X 0,Y 235.712,Z 257.586,A -85,B 0,C 180,E1 -19545.12,E2 -19545.12} C_VEL
LIN {X 0,Y 236.313,Z 248.299,A -85,B 0,C 180,E1 -19546.408,E2 -19546.408} C_VEL
LIN {X 0,Y 235.402,Z 237.357,A -85,B 0,C 180,E1 -19547.592,E2 -19547.592} C_VEL
LIN {X 0,Y 234.581,Z 224.631,A -85,B 0,C 180,E1 -19548.615,E2 -19548.615} C_VEL
LIN {X 0,Y 234.567,Z 219.847,A -85,B 0,C 180,E1 -19548.956,E2 -19548.956} C_VEL
LIN {X 0,Y 236.233,Z 209.181,A -85,B 0,C 180,E1 -19554.611,E2 -19554.611} C_VEL
LIN {X 0,Y 238.124,Z 200.567,A -85,B 0,C 180,E1 -19559.139,E2 -19559.139} C_VEL
LIN {X 0,Y 237.733,Z 197.191,A -85,B 0,C 180,E1 -19560.983,E2 -19560.983} C_VEL
LIN {X 0,Y 235.779,Z 187.331,A -85,B 0,C 180,E1 -19566.591,E2 -19566.591} C_VEL
LIN {X 0,Y 235.007,Z 183.208,A -85,B 0,C 180,E1 -19569.054,E2 -19569.054} C_VEL
LIN {X 0,Y 234.898,Z 183.225,A -85,B 0,C 180,E1 -19574.105,E2 -19574.105} C_VEL
LIN {X 0,Y 234.951,Z 183.218,A -85,B 0,C 180,E1 -19578.397,E2 -19578.397} C_VEL
LIN {X 0,Y 234.946,Z 183.217,A -85,B 0,C 180,E1 -19581.084,E2 -19581.084} C_VEL
LIN {X 0,Y 234.951,Z 183.214,A -85,B 0,C 180,E1 -19585.365,E2 -19585.365} C_VEL
LIN {X 0,Y 234.912,Z 183.222,A -85,B 0,C 180,E1 -19589.429,E2 -19589.429} C_VEL
LIN {X 0,Y 234.982,Z 183.214,A -85,B 0,C 180,E1 -19593.792,E2 -19593.792} C_VEL
LIN {X 0,Y 234.986,Z 183.212,A -85,B 0,C 180,E1 -19598.967,E2 -19598.967} C_VEL
LIN {X 0,Y 235.084,Z 183.198,A -85,B 0,C 180,E1 -19603.058,E2 -19603.058} C_VEL
LIN {X 0,Y 235.134,Z 183.194,A -85,B 0,C 180,E1 -19607.923,E2 -19607.923} C_VEL
LIN {X 0,Y 235.363,Z 183.166,A -85,B 0,C 180,E1 -19611.413,E2 -19611.413} C_VEL
LIN {X 0,Y 235.39,Z 183.163,A -85,B 0,C 180,E1 -19613.141,E2 -19613.141} C_VEL
LIN {X 0,Y 235.586,Z 183.137,A -85,B 0,C 180,E1 -19618.29,E2 -19618.29} C_VEL
LIN {X 0,Y 235.581,Z 183.137,A -85,B 0,C 180,E1 -19621.709,E2 -19621.709} C_VEL
LIN {X 0,Y 235.39,Z 183.163,A -85,B 0,C 180,E1 -19626.859,E2 -19626.859} C_VEL
LIN {X 0,Y 235.225,Z 183.182,A -85,B 0,C 180,E1 -19630.327,E2 -19630.327} C_VEL
LIN {X 0,Y 235.101,Z 183.197,A -85,B 0,C 180,E1 -19635.607,E2 -19635.607} C_VEL
LIN {X 0,Y 234.996,Z 183.21,A -85,B 0,C 180,E1 -19639.207,E2 -19639.207} C_VEL
LIN {X 0,Y 234.936,Z 183.218,A -85,B 0,C 180,E1 -19642.885,E2 -19642.885} C_VEL
LIN {X 0,Y 234.934,Z 183.218,A -85,B 0,C 180,E1 -19646.662,E2 -19646.662} C_VEL
LIN {X 0,Y 234.888,Z 183.225,A -85,B 0,C 180,E1 -19650.574,E2 -19650.574} C_VEL
LIN {X 0,Y 234.949,Z 183.214,A -85,B 0,C 180,E1 -19654.635,E2 -19654.635} C_VEL
LIN {X 0,Y 234.932,Z 183.219,A -85,B 0,C 180,E1 -19658.946,E2 -19658.946} C_VEL
LIN {X 0,Y 234.913,Z 183.222,A -85,B 0,C 180,E1 -19663.48,E2 -19663.48} C_VEL
LIN {X 0,Y 234.882,Z 183.225,A -85,B 0,C 180,E1 -19666.517,E2 -19666.517} C_VEL
LIN {X 0,Y 234.911,Z 183.222,A -85,B 0,C 180,E1 -19671.081,E2 -19671.081} C_VEL
LIN {X 0,Y 234.924,Z 183.223,A -85,B 0,C 180,E1 -19675.365,E2 -19675.365} C_VEL
LIN {X 0,Y 234.926,Z 183.218,A -85,B 0,C 180,E1 -19679.435,E2 -19679.435} C_VEL
LIN {X 0,Y 234.99,Z 183.212,A -85,B 0,C 180,E1 -19683.796,E2 -19683.796} C_VEL
LIN {X 0,Y 235.008,Z 183.21,A -85,B 0,C 180,E1 -19688.973,E2 -19688.973} C_VEL
LIN {X 0,Y 235.094,Z 183.2,A -85,B 0,C 180,E1 -19693.062,E2 -19693.062} C_VEL
LIN {X 0,Y 235.117,Z 183.194,A -85,B 0,C 180,E1 -19697.925,E2 -19697.925} C_VEL
LIN {X 0,Y 235.39,Z 183.162,A -85,B 0,C 180,E1 -19701.417,E2 -19701.417} C_VEL
LIN {X 0,Y 235.406,Z 183.159,A -85,B 0,C 180,E1 -19703.144,E2 -19703.144} C_VEL
LIN {X 0,Y 235.594,Z 183.139,A -85,B 0,C 180,E1 -19708.293,E2 -19708.293} C_VEL
LIN {X 0,Y 235.592,Z 183.139,A -85,B 0,C 180,E1 -19711.712,E2 -19711.712} C_VEL
LIN {X 0,Y 235.408,Z 183.159,A -85,B 0,C 180,E1 -19716.861,E2 -19716.861} C_VEL
LIN {X 0,Y 235.257,Z 183.178,A -85,B 0,C 180,E1 -19720.328,E2 -19720.328} C_VEL
LIN {X 0,Y 235.118,Z 183.199,A -85,B 0,C 180,E1 -19725.609,E2 -19725.609} C_VEL
LIN {X 0,Y 235.008,Z 183.212,A -85,B 0,C 180,E1 -19729.208,E2 -19729.208} C_VEL
LIN {X 0,Y 234.921,Z 183.22,A -85,B 0,C 180,E1 -19732.89,E2 -19732.89} C_VEL
LIN {X 0,Y 234.93,Z 183.22,A -85,B 0,C 180,E1 -19736.665,E2 -19736.665} C_VEL
LIN {X 0,Y 234.904,Z 183.221,A -85,B 0,C 180,E1 -19740.574,E2 -19740.574} C_VEL
LIN {X 0,Y 234.934,Z 183.221,A -85,B 0,C 180,E1 -19744.64,E2 -19744.64} C_VEL
LIN {X 0,Y 234.917,Z 183.221,A -85,B 0,C 180,E1 -19748.937,E2 -19748.937} C_VEL
LIN {X 0,Y 234.872,Z 183.226,A -85,B 0,C 180,E1 -19753.493,E2 -19753.493} C_VEL
LIN {X 0,Y 234.892,Z 183.224,A -85,B 0,C 180,E1 -19756.515,E2 -19756.515} C_VEL
LIN {X 0,Y 234.962,Z 183.215,A -85,B 0,C 180,E1 -19761.087,E2 -19761.087} C_VEL
LIN {X 0,Y 235.166,Z 183.239,A -85,B 0,C 180,E1 -19764.618,E2 -19764.618} C_VEL
LIN {X 0,Y 235.909,Z 187.343,A -85,B 0,C 180,E1 -19767.572,E2 -19767.572} C_VEL
LIN {X 0,Y 235.957,Z 190.47,A -85,B 0,C 180,E1 -19769.746,E2 -19769.746} C_VEL
LIN {X 0,Y 234.981,Z 197.426,A -85,B 0,C 180,E1 -19774.478,E2 -19774.478} C_VEL
LIN {X 0,Y 234.267,Z 204.02,A -85,B 0,C 180,E1 -19778.9,E2 -19778.9} C_VEL
LIN {X 0,Y 233.606,Z 210.793,A -85,B 0,C 180,E1 -19783.393,E2 -19783.393} C_VEL
LIN {X 0,Y 233.409,Z 217.102,A -85,B 0,C 180,E1 -19787.557,E2 -19787.557} C_VEL
LIN {X 0,Y 234.013,Z 228.983,A -85,B 0,C 180,E1 -19788.743,E2 -19788.743} C_VEL
LIN {X 0,Y 234.716,Z 237.973,A -85,B 0,C 180,E1 -19789.868,E2 -19789.868} C_VEL
LIN {X 0,Y 234.218,Z 248.754,A -85,B 0,C 180,E1 -19791.589,E2 -19791.589} C_VEL
LIN {X 0,Y 233.684,Z 258.53,A -85,B 0,C 180,E1 -19793.577,E2 -19793.577} C_VEL
LIN {X 0,Y 233.471,Z 266.849,A -85,B 0,C 180,E1 -19795.684,E2 -19795.684} C_VEL
LIN {X 0,Y 233.095,Z 273.615,A -85,B 0,C 180,E1 -19797.84,E2 -19797.84} C_VEL
LIN {X 0,Y 232.985,Z 279.045,A -85,B 0,C 180,E1 -19800,E2 -19800} C_VEL
LIN {X 0,Y 233.289,Z 284.058,A -85,B 0,C 180,E1 -19802.59,E2 -19802.59} C_VEL
LIN {X 0,Y 234.067,Z 287.662,A -85,B 0,C 180,E1 -19805.168,E2 -19805.168} C_VEL
LIN {X 0,Y 234.873,Z 289.332,A -85,B 0,C 180,E1 -19806.874,E2 -19806.874} C_VEL
LIN {X 0,Y 235.642,Z 290.428,A -85,B 0,C 180,E1 -19808.576,E2 -19808.576} C_VEL
LIN {X 0,Y 236.765,Z 291.011,A -85,B 0,C 180,E1 -19810.259,E2 -19810.259} C_VEL
LIN {X 0,Y 238.139,Z 291.048,A -85,B 0,C 180,E1 -19811.922,E2 -19811.922} C_VEL
LIN {X 0,Y 239.912,Z 290.524,A -85,B 0,C 180,E1 -19813.554,E2 -19813.554} C_VEL
LIN {X 0,Y 241.735,Z 289.528,A -85,B 0,C 180,E1 -19815.169,E2 -19815.169} C_VEL
LIN {X 0,Y 245.128,Z 286.96,A -85,B 0,C 180,E1 -19817.52,E2 -19817.52} C_VEL
LIN {X 0,Y 249.048,Z 283.14,A -85,B 0,C 180,E1 -19819.794,E2 -19819.794} C_VEL
LIN {X 0,Y 253.333,Z 278.014,A -85,B 0,C 180,E1 -19821.995,E2 -19821.995} C_VEL
LIN {X 0,Y 254.77,Z 276.021,A -85,B 0,C 180,E1 -19822.718,E2 -19822.718} C_VEL
LIN {X 0,Y 256.82,Z 270.973,A -85,B 0,C 180,E1 -19824.781,E2 -19824.781} C_VEL
LIN {X 0,Y 258.491,Z 264.168,A -85,B 0,C 180,E1 -19827.53,E2 -19827.53} C_VEL
LIN {X 0,Y 259.444,Z 257.359,A -85,B 0,C 180,E1 -19830.401,E2 -19830.401} C_VEL
LIN {X 0,Y 259.891,Z 251.729,A -85,B 0,C 180,E1 -19833.035,E2 -19833.035} C_VEL
LIN {X 0,Y 259.941,Z 248.96,A -85,B 0,C 180,E1 -19834.595,E2 -19834.595} C_VEL
LIN {X 0,Y 259.643,Z 246.52,A -85,B 0,C 180,E1 -19836.548,E2 -19836.548} C_VEL
LIN {X 0,Y 259.441,Z 244.737,A -85,B 0,C 180,E1 -19838.539,E2 -19838.539} C_VEL
LIN {X 0,Y 259.187,Z 243.914,A -85,B 0,C 180,E1 -19840.6,E2 -19840.6} C_VEL
LIN {X 0,Y 259.258,Z 243.767,A -85,B 0,C 180,E1 -19842.95,E2 -19842.95} C_VEL
LIN {X 0,Y 259.81,Z 244.333,A -85,B 0,C 180,E1 -19845.304,E2 -19845.304} C_VEL
LIN {X 0,Y 260.743,Z 245.751,A -85,B 0,C 180,E1 -19847.633,E2 -19847.633} C_VEL
LIN {X 0,Y 261.014,Z 246.559,A -85,B 0,C 180,E1 -19848.36,E2 -19848.36} C_VEL
LIN {X 0,Y 261.336,Z 248.407,A -85,B 0,C 180,E1 -19849.601,E2 -19849.601} C_VEL
LIN {X 0,Y 261.32,Z 250.961,A -85,B 0,C 180,E1 -19850.785,E2 -19850.785} C_VEL
LIN {X 0,Y 261.147,Z 252.945,A -85,B 0,C 180,E1 -19851.543,E2 -19851.543} C_VEL
LIN {X 0,Y 260.485,Z 257.389,A -85,B 0,C 180,E1 -19853.017,E2 -19853.017} C_VEL
LIN {X 0,Y 259.562,Z 262.096,A -85,B 0,C 180,E1 -19854.45,E2 -19854.45} C_VEL
LIN {X 0,Y 257.422,Z 270.516,A -85,B 0,C 180,E1 -19856.902,E2 -19856.902} C_VEL
LIN {X 0,Y 255.24,Z 276.206,A -85,B 0,C 180,E1 -19858.453,E2 -19858.453} C_VEL
LIN {X 0,Y 249.885,Z 284.598,A -85,B 0,C 180,E1 -19860.513,E2 -19860.513} C_VEL
LIN {X 0,Y 244.911,Z 291.55,A -85,B 0,C 180,E1 -19862.666,E2 -19862.666} C_VEL
LIN {X 0,Y 240.014,Z 297.809,A -85,B 0,C 180,E1 -19865.194,E2 -19865.194} C_VEL
LIN {X 0,Y 236.562,Z 301.832,A -85,B 0,C 180,E1 -19867.278,E2 -19867.278} C_VEL
LIN {X 0,Y 232.618,Z 306.458,A -85,B 0,C 180,E1 -19870.587,E2 -19870.587} C_VEL
LIN {X 0,Y 229.317,Z 309.524,A -85,B 0,C 180,E1 -19873.986,E2 -19873.986} C_VEL
LIN {X 0,Y 228.082,Z 310.52,A -85,B 0,C 180,E1 -19875.726,E2 -19875.726} C_VEL
LIN {X 0,Y 226.614,Z 311.382,A -85,B 0,C 180,E1 -19879.273,E2 -19879.273} C_VEL
LIN {X 0,Y 225.986,Z 310.82,A -85,B 0,C 180,E1 -19882.851,E2 -19882.851} C_VEL
LIN {X 0,Y 226.061,Z 309.966,A -85,B 0,C 180,E1 -19884.646,E2 -19884.646} C_VEL
LIN {X 0,Y 226.53,Z 307.078,A -85,B 0,C 180,E1 -19888.219,E2 -19888.219} C_VEL
LIN {X 0,Y 226.885,Z 303.662,A -85,B 0,C 180,E1 -19890.885,E2 -19890.885} C_VEL
LIN {X 0,Y 226.866,Z 298.92,A -85,B 0,C 180,E1 -19893.549,E2 -19893.549} C_VEL
LIN {X 0,Y 226.978,Z 292.779,A -85,B 0,C 180,E1 -19896.219,E2 -19896.219} C_VEL
LIN {X 0,Y 227.056,Z 286.457,A -85,B 0,C 180,E1 -19898.403,E2 -19898.403} C_VEL
LIN {X 0,Y 227.415,Z 278.406,A -85,B 0,C 180,E1 -19900.683,E2 -19900.683} C_VEL
LIN {X 0,Y 227.935,Z 268.612,A -85,B 0,C 180,E1 -19902.914,E2 -19902.914} C_VEL
LIN {X 0,Y 228.539,Z 258.906,A -85,B 0,C 180,E1 -19904.694,E2 -19904.694} C_VEL
LIN {X 0,Y 229.237,Z 248.475,A -85,B 0,C 180,E1 -19906.221,E2 -19906.221} C_VEL
LIN {X 0,Y 228.358,Z 237.778,A -85,B 0,C 180,E1 -19907.433,E2 -19907.433} C_VEL
LIN {X 0,Y 227.514,Z 224.991,A -85,B 0,C 180,E1 -19908.514,E2 -19908.514} C_VEL
LIN {X 0,Y 227.48,Z 219.921,A -85,B 0,C 180,E1 -19908.867,E2 -19908.867} C_VEL
LIN {X 0,Y 229.048,Z 209.701,A -85,B 0,C 180,E1 -19914.467,E2 -19914.467} C_VEL
LIN {X 0,Y 230.988,Z 201.161,A -85,B 0,C 180,E1 -19919.128,E2 -19919.128} C_VEL
LIN {X 0,Y 230.58,Z 197.485,A -85,B 0,C 180,E1 -19921.205,E2 -19921.205} C_VEL
LIN {X 0,Y 228.859,Z 188.797,A -85,B 0,C 180,E1 -19926.292,E2 -19926.292} C_VEL
LIN {X 0,Y 227.967,Z 184.084,A -85,B 0,C 180,E1 -19929.185,E2 -19929.185} C_VEL
LIN {X 0,Y 227.842,Z 184.103,A -85,B 0,C 180,E1 -19934.809,E2 -19934.809} C_VEL
LIN {X 0,Y 227.901,Z 184.092,A -85,B 0,C 180,E1 -19937.736,E2 -19937.736} C_VEL
LIN {X 0,Y 227.862,Z 184.101,A -85,B 0,C 180,E1 -19941.912,E2 -19941.912} C_VEL
LIN {X 0,Y 227.881,Z 184.098,A -85,B 0,C 180,E1 -19946.371,E2 -19946.371} C_VEL
LIN {X 0,Y 227.894,Z 184.097,A -85,B 0,C 180,E1 -19950.434,E2 -19950.434} C_VEL
LIN {X 0,Y 227.913,Z 184.091,A -85,B 0,C 180,E1 -19954.424,E2 -19954.424} C_VEL
LIN {X 0,Y 227.936,Z 184.091,A -85,B 0,C 180,E1 -19958.284,E2 -19958.284} C_VEL
LIN {X 0,Y 228.022,Z 184.077,A -85,B 0,C 180,E1 -19962.825,E2 -19962.825} C_VEL
LIN {X 0,Y 228.082,Z 184.075,A -85,B 0,C 180,E1 -19967.544,E2 -19967.544} C_VEL
LIN {X 0,Y 228.293,Z 184.047,A -85,B 0,C 180,E1 -19971.145,E2 -19971.145} C_VEL
LIN {X 0,Y 228.341,Z 184.04,A -85,B 0,C 180,E1 -19972.928,E2 -19972.928} C_VEL
LIN {X 0,Y 228.545,Z 184.014,A -85,B 0,C 180,E1 -19978.238,E2 -19978.238} C_VEL
LIN {X 0,Y 228.54,Z 184.014,A -85,B 0,C 180,E1 -19981.762,E2 -19981.762} C_VEL
LIN {X 0,Y 228.342,Z 184.04,A -85,B 0,C 180,E1 -19987.072,E2 -19987.072} C_VEL
LIN {X 0,Y 228.151,Z 184.066,A -85,B 0,C 180,E1 -19990.651,E2 -19990.651} C_VEL
LIN {X 0,Y 228.052,Z 184.078,A -85,B 0,C 180,E1 -19994.273,E2 -19994.273} C_VEL
LIN {X 0,Y 227.991,Z 184.082,A -85,B 0,C 180,E1 -19997.954,E2 -19997.954} C_VEL
LIN {X 0,Y 227.91,Z 184.097,A -85,B 0,C 180,E1 -20002.326,E2 -20002.326} C_VEL
LIN {X 0,Y 227.911,Z 184.093,A -85,B 0,C 180,E1 -20006.594,E2 -20006.594} C_VEL
LIN {X 0,Y 227.862,Z 184.101,A -85,B 0,C 180,E1 -20010.283,E2 -20010.283} C_VEL
LIN {X 0,Y 227.878,Z 184.099,A -85,B 0,C 180,E1 -20013.72,E2 -20013.72} C_VEL
LIN {X 0,Y 227.86,Z 184.102,A -85,B 0,C 180,E1 -20018.088,E2 -20018.088} C_VEL
LIN {X 0,Y 227.838,Z 184.1,A -85,B 0,C 180,E1 -20022.736,E2 -20022.736} C_VEL
LIN {X 0,Y 227.805,Z 184.11,A -85,B 0,C 180,E1 -20027.261,E2 -20027.261} C_VEL
LIN {X 0,Y 227.836,Z 184.101,A -85,B 0,C 180,E1 -20031.912,E2 -20031.912} C_VEL
LIN {X 0,Y 227.873,Z 184.099,A -85,B 0,C 180,E1 -20036.38,E2 -20036.38} C_VEL
LIN {X 0,Y 227.914,Z 184.09,A -85,B 0,C 180,E1 -20040.441,E2 -20040.441} C_VEL
LIN {X 0,Y 227.925,Z 184.093,A -85,B 0,C 180,E1 -20044.429,E2 -20044.429} C_VEL
LIN {X 0,Y 227.959,Z 184.087,A -85,B 0,C 180,E1 -20048.29,E2 -20048.29} C_VEL
LIN {X 0,Y 228.033,Z 184.081,A -85,B 0,C 180,E1 -20052.828,E2 -20052.828} C_VEL
LIN {X 0,Y 228.074,Z 184.07,A -85,B 0,C 180,E1 -20057.546,E2 -20057.546} C_VEL
LIN {X 0,Y 228.325,Z 184.042,A -85,B 0,C 180,E1 -20061.15,E2 -20061.15} C_VEL
LIN {X 0,Y 228.359,Z 184.038,A -85,B 0,C 180,E1 -20062.932,E2 -20062.932} C_VEL
LIN {X 0,Y 228.553,Z 184.016,A -85,B 0,C 180,E1 -20068.241,E2 -20068.241} C_VEL
LIN {X 0,Y 228.552,Z 184.016,A -85,B 0,C 180,E1 -20071.765,E2 -20071.765} C_VEL
LIN {X 0,Y 228.361,Z 184.037,A -85,B 0,C 180,E1 -20077.074,E2 -20077.074} C_VEL
LIN {X 0,Y 228.171,Z 184.06,A -85,B 0,C 180,E1 -20080.653,E2 -20080.653} C_VEL
LIN {X 0,Y 228.069,Z 184.073,A -85,B 0,C 180,E1 -20084.274,E2 -20084.274} C_VEL
LIN {X 0,Y 228.006,Z 184.082,A -85,B 0,C 180,E1 -20087.956,E2 -20087.956} C_VEL
LIN {X 0,Y 227.909,Z 184.092,A -85,B 0,C 180,E1 -20092.316,E2 -20092.316} C_VEL
LIN {X 0,Y 227.907,Z 184.095,A -85,B 0,C 180,E1 -20096.584,E2 -20096.584} C_VEL
LIN {X 0,Y 227.878,Z 184.094,A -85,B 0,C 180,E1 -20100.283,E2 -20100.283} C_VEL
LIN {X 0,Y 227.882,Z 184.097,A -85,B 0,C 180,E1 -20103.722,E2 -20103.722} C_VEL
LIN {X 0,Y 227.849,Z 184.099,A -85,B 0,C 180,E1 -20108.093,E2 -20108.093} C_VEL
LIN {X 0,Y 227.799,Z 184.11,A -85,B 0,C 180,E1 -20112.748,E2 -20112.748} C_VEL
LIN {X 0,Y 227.82,Z 184.102,A -85,B 0,C 180,E1 -20117.26,E2 -20117.26} C_VEL
LIN {X 0,Y 227.928,Z 184.093,A -85,B 0,C 180,E1 -20121.926,E2 -20121.926} C_VEL
LIN {X 0,Y 228.161,Z 184.231,A -85,B 0,C 180,E1 -20124.697,E2 -20124.697} C_VEL
LIN {X 0,Y 228.998,Z 189.462,A -85,B 0,C 180,E1 -20128.552,E2 -20128.552} C_VEL
LIN {X 0,Y 228.272,Z 195.086,A -85,B 0,C 180,E1 -20132.496,E2 -20132.496} C_VEL
LIN {X 0,Y 227.403,Z 201.992,A -85,B 0,C 180,E1 -20137.275,E2 -20137.275} C_VEL
LIN {X 0,Y 226.716,Z 208.789,A -85,B 0,C 180,E1 -20141.941,E2 -20141.941} C_VEL
LIN {X 0,Y 226.319,Z 217.136,A -85,B 0,C 180,E1 -20147.616,E2 -20147.616} C_VEL
LIN {X 0,Y 227.067,Z 230.809,A -85,B 0,C 180,E1 -20149.072,E2 -20149.072} C_VEL
LIN {X 0,Y 227.623,Z 237.848,A -85,B 0,C 180,E1 -20149.999,E2 -20149.999} C_VEL
LIN {X 0,Y 227.109,Z 248.968,A -85,B 0,C 180,E1 -20151.832,E2 -20151.832} C_VEL
LIN {X 0,Y 226.634,Z 258.193,A -85,B 0,C 180,E1 -20153.752,E2 -20153.752} C_VEL
LIN {X 0,Y 226.389,Z 266.826,A -85,B 0,C 180,E1 -20155.995,E2 -20155.995} C_VEL
LIN {X 0,Y 226.022,Z 273.654,A -85,B 0,C 180,E1 -20158.218,E2 -20158.218} C_VEL
LIN {X 0,Y 225.967,Z 280.094,A -85,B 0,C 180,E1 -20160.891,E2 -20160.891} C_VEL
LIN {X 0,Y 226.433,Z 284.937,A -85,B 0,C 180,E1 -20163.559,E2 -20163.559} C_VEL
LIN {X 0,Y 227.021,Z 287.39,A -85,B 0,C 180,E1 -20165.329,E2 -20165.329} C_VEL
LIN {X 0,Y 227.845,Z 289.269,A -85,B 0,C 180,E1 -20167.087,E2 -20167.087} C_VEL
LIN {X 0,Y 228.653,Z 290.603,A -85,B 0,C 180,E1 -20168.841,E2 -20168.841} C_VEL
LIN {X 0,Y 229.811,Z 291.381,A -85,B 0,C 180,E1 -20170.573,E2 -20170.573} C_VEL
LIN {X 0,Y 231.225,Z 291.661,A -85,B 0,C 180,E1 -20172.284,E2 -20172.284} C_VEL
LIN {X 0,Y 233.084,Z 291.378,A -85,B 0,C 180,E1 -20173.959,E2 -20173.959} C_VEL
LIN {X 0,Y 234.973,Z 290.603,A -85,B 0,C 180,E1 -20175.616,E2 -20175.616} C_VEL
LIN {X 0,Y 237.229,Z 289.313,A -85,B 0,C 180,E1 -20177.233,E2 -20177.233} C_VEL
LIN {X 0,Y 241.174,Z 286.313,A -85,B 0,C 180,E1 -20179.58,E2 -20179.58} C_VEL
LIN {X 0,Y 245.463,Z 282.121,A -85,B 0,C 180,E1 -20181.852,E2 -20181.852} C_VEL
LIN {X 0,Y 248.541,Z 278.598,A -85,B 0,C 180,E1 -20183.321,E2 -20183.321} C_VEL
LIN {X 0,Y 250.504,Z 275.03,A -85,B 0,C 180,E1 -20184.887,E2 -20184.887} C_VEL
LIN {X 0,Y 252.497,Z 269.577,A -85,B 0,C 180,E1 -20187.339,E2 -20187.339} C_VEL
LIN {X 0,Y 253.961,Z 263.94,A -85,B 0,C 180,E1 -20189.876,E2 -20189.876} C_VEL
LIN {X 0,Y 254.986,Z 258.446,A -85,B 0,C 180,E1 -20192.543,E2 -20192.543} C_VEL
LIN {X 0,Y 255.412,Z 255.244,A -85,B 0,C 180,E1 -20194.359,E2 -20194.359} C_VEL
LIN {X 0,Y 255.489,Z 253.872,A -85,B 0,C 180,E1 -20195.287,E2 -20195.287} C_VEL
LIN {X 0,Y 255.465,Z 251.748,A -85,B 0,C 180,E1 -20197.246,E2 -20197.246} C_VEL
LIN {X 0,Y 255.356,Z 250.243,A -85,B 0,C 180,E1 -20199.587,E2 -20199.587} C_VEL
LIN {X 0,Y 255.355,Z 249.767,A -85,B 0,C 180,E1 -20202,E2 -20202} C_VEL
LIN {X 0,Y 256.066,Z 250.443,A -85,B 0,C 180,E1 -20205.529,E2 -20205.529} C_VEL
LIN {X 0,Y 256.84,Z 251.774,A -85,B 0,C 180,E1 -20207.631,E2 -20207.631} C_VEL
LIN {X 0,Y 258.147,Z 255.233,A -85,B 0,C 180,E1 -20210.709,E2 -20210.709} C_VEL
LIN {X 0,Y 259.34,Z 259.755,A -85,B 0,C 180,E1 -20213.4,E2 -20213.4} C_VEL
LIN {X 0,Y 259.677,Z 261.551,A -85,B 0,C 180,E1 -20214.285,E2 -20214.285} C_VEL
LIN {X 0,Y 259.562,Z 262.096,A -85,B 0,C 180,E1 -20214.45,E2 -20214.45} C_VEL
LIN {X 0,Y 258.229,Z 266,A -85,B 0,C 180,E1 -20215.413,E2 -20215.413} C_VEL
LIN {X 0,Y 255.979,Z 270.198,A -85,B 0,C 180,E1 -20216.226,E2 -20216.226} C_VEL
LIN {X 0,Y 248.04,Z 281.121,A -85,B 0,C 180,E1 -20218.244,E2 -20218.244} C_VEL
LIN {X 0,Y 246.162,Z 283.563,A -85,B 0,C 180,E1 -20218.844,E2 -20218.844} C_VEL
LIN {X 0,Y 240.431,Z 291.055,A -85,B 0,C 180,E1 -20221.161,E2 -20221.161} C_VEL
LIN {X 0,Y 234.613,Z 297.813,A -85,B 0,C 180,E1 -20223.942,E2 -20223.942} C_VEL
LIN {X 0,Y 230.074,Z 302.57,A -85,B 0,C 180,E1 -20226.6,E2 -20226.6} C_VEL
LIN {X 0,Y 225.927,Z 306.747,A -85,B 0,C 180,E1 -20229.987,E2 -20229.987} C_VEL
LIN {X 0,Y 222.495,Z 309.439,A -85,B 0,C 180,E1 -20233.481,E2 -20233.481} C_VEL
LIN {X 0,Y 220.288,Z 310.71,A -85,B 0,C 180,E1 -20237.093,E2 -20237.093} C_VEL
LIN {X 0,Y 219.167,Z 310.526,A -85,B 0,C 180,E1 -20240.771,E2 -20240.771} C_VEL
LIN {X 0,Y 219.065,Z 308.936,A -85,B 0,C 180,E1 -20244.474,E2 -20244.474} C_VEL
LIN {X 0,Y 219.558,Z 305.713,A -85,B 0,C 180,E1 -20248.163,E2 -20248.163} C_VEL
LIN {X 0,Y 219.882,Z 303.433,A -85,B 0,C 180,E1 -20249.997,E2 -20249.997} C_VEL
LIN {X 0,Y 219.94,Z 298.877,A -85,B 0,C 180,E1 -20252.744,E2 -20252.744} C_VEL
LIN {X 0,Y 220.012,Z 292.885,A -85,B 0,C 180,E1 -20255.496,E2 -20255.496} C_VEL
LIN {X 0,Y 220.105,Z 286.262,A -85,B 0,C 180,E1 -20257.909,E2 -20257.909} C_VEL
LIN {X 0,Y 220.342,Z 278.915,A -85,B 0,C 180,E1 -20260.1,E2 -20260.1} C_VEL
LIN {X 0,Y 220.82,Z 269.375,A -85,B 0,C 180,E1 -20262.403,E2 -20262.403} C_VEL
LIN {X 0,Y 221.47,Z 258.642,A -85,B 0,C 180,E1 -20264.468,E2 -20264.468} C_VEL
LIN {X 0,Y 222.185,Z 248.169,A -85,B 0,C 180,E1 -20266.065,E2 -20266.065} C_VEL
LIN {X 0,Y 221.237,Z 237.221,A -85,B 0,C 180,E1 -20267.342,E2 -20267.342} C_VEL
LIN {X 0,Y 220.442,Z 224.152,A -85,B 0,C 180,E1 -20268.477,E2 -20268.477} C_VEL
